LIN {X 86.419,Y -41.764,Z -98.944,A -90.000,B 90.000,C 0.000} C_DIS
LIN {X 86.321,Y -41.760,Z -99.036,A -90.000,B 90.000,C 0.000} C_DIS
LIN {X 86.213,Y -41.757,Z -99.132,A -90.000,B 90.000,C 0.000} C_DIS
LIN {X 85.903,Y -41.758,Z -99.390,A -90.000,B 90.000,C 0.000} C_DIS
LIN {X 85.446,Y -41.767,Z -99.745,A -90.000,B 90.000,C 0.000} C_DIS
LIN {X 85.305,Y -41.778,Z -99.859,A -90.000,B 90.000,C 0.000} C_DIS
LIN {X 85.131,Y -41.796,Z -99.993,A -90.000,B 90.000,C 0.000} C_DIS
LIN {X 84.957,Y -41.819,Z -100.115,A -90.000,B 90.000,C 0.000} C_DIS
LIN {X 84.802,Y -41.842,Z -100.215,A -90.000,B 90.000,C 0.000} C_DIS
LIN {X 84.683,Y -41.862,Z -100.286,A -90.000,B 90.000,C 0.000} C_DIS
LIN {X 84.481,Y -41.884,Z -100.395,A -90.000,B 90.000,C 0.000} C_DIS
LIN {X 84.221,Y -41.928,Z -100.537,A -90.000,B 90.000,C 0.000} C_DIS
LIN {X 84.067,Y -41.950,Z -100.619,A -90.000,B 90.000,C 0.000} C_DIS
LIN {X 83.579,Y -42.021,Z -100.876,A -90.000,B 90.000,C 0.000} C_DIS
LIN {X 83.391,Y -42.049,Z -100.970,A -90.000,B 90.000,C 0.000} C_DIS
LIN {X 83.264,Y -42.075,Z -101.035,A -90.000,B 90.000,C 0.000} C_DIS
LIN {X 82.879,Y -42.146,Z -101.260,A -90.000,B 90.000,C 0.000} C_DIS
LIN {X 82.672,Y -42.176,Z -101.400,A -90.000,B 90.000,C 0.000} C_DIS
LIN {X 82.594,Y -42.188,Z -101.451,A -90.000,B 90.000,C 0.000} C_DIS
LIN {X 82.374,Y -42.226,Z -101.578,A -90.000,B 90.000,C 0.000} C_DIS
LIN {X 82.222,Y -42.254,Z -101.660,A -90.000,B 90.000,C 0.000} C_DIS
LIN {X 82.012,Y -42.297,Z -101.771,A -90.000,B 90.000,C 0.000} C_DIS
LIN {X 81.894,Y -42.322,Z -101.825,A -90.000,B 90.000,C 0.000} C_DIS
LIN {X 81.742,Y -42.355,Z -101.888,A -90.000,B 90.000,C 0.000} C_DIS
LIN {X 81.659,Y -42.371,Z -101.920,A -90.000,B 90.000,C 0.000} C_DIS
LIN {X 81.529,Y -42.394,Z -101.964,A -90.000,B 90.000,C 0.000} C_DIS
LIN {X 81.072,Y -42.475,Z -102.099,A -90.000,B 90.000,C 0.000} C_DIS
LIN {X 81.028,Y -42.482,Z -102.115,A -90.000,B 90.000,C 0.000} C_DIS
LIN {X 80.881,Y -42.501,Z -102.170,A -90.000,B 90.000,C 0.000} C_DIS
LIN {X 80.690,Y -42.524,Z -102.247,A -90.000,B 90.000,C 0.000} C_DIS
LIN {X 80.320,Y -42.591,Z -102.396,A -90.000,B 90.000,C 0.000} C_DIS
LIN {X 79.816,Y -42.684,Z -102.594,A -90.000,B 90.000,C 0.000} C_DIS
LIN {X 79.637,Y -42.717,Z -102.663,A -90.000,B 90.000,C 0.000} C_DIS
LIN {X 79.531,Y -42.736,Z -102.698,A -90.000,B 90.000,C 0.000} C_DIS
LIN {X 79.408,Y -42.759,Z -102.750,A -90.000,B 90.000,C 0.000} C_DIS
LIN {X 79.279,Y -42.782,Z -102.801,A -90.000,B 90.000,C 0.000} C_DIS
LIN {X 79.059,Y -42.822,Z -102.874,A -90.000,B 90.000,C 0.000} C_DIS
LIN {X 78.928,Y -42.846,Z -102.910,A -90.000,B 90.000,C 0.000} C_DIS
LIN {X 78.902,Y -42.851,Z -102.916,A -90.000,B 90.000,C 0.000} C_DIS
LIN {X 78.691,Y -42.870,Z -102.962,A -90.000,B 90.000,C 0.000} C_DIS
LIN {X 78.445,Y -42.891,Z -103.005,A -90.000,B 90.000,C 0.000} C_DIS
LIN {X 78.333,Y -42.900,Z -103.021,A -90.000,B 90.000,C 0.000} C_DIS
LIN {X 78.121,Y -42.912,Z -103.046,A -90.000,B 90.000,C 0.000} C_DIS
LIN {X 77.986,Y -42.919,Z -103.054,A -90.000,B 90.000,C 0.000} C_DIS
LIN {X 77.768,Y -42.931,Z -103.059,A -90.000,B 90.000,C 0.000} C_DIS
LIN {X 77.616,Y -42.940,Z -103.055,A -90.000,B 90.000,C 0.000} C_DIS
LIN {X 77.437,Y -42.949,Z -103.044,A -90.000,B 90.000,C 0.000} C_DIS
LIN {X 77.279,Y -42.957,Z -103.028,A -90.000,B 90.000,C 0.000} C_DIS
LIN {X 77.030,Y -42.970,Z -102.997,A -90.000,B 90.000,C 0.000} C_DIS
LIN {X 76.845,Y -42.979,Z -102.965,A -90.000,B 90.000,C 0.000} C_DIS
LIN {X 76.645,Y -42.989,Z -102.921,A -90.000,B 90.000,C 0.000} C_DIS
LIN {X 76.463,Y -43.002,Z -102.870,A -90.000,B 90.000,C 0.000} C_DIS
LIN {X 76.351,Y -43.011,Z -102.835,A -90.000,B 90.000,C 0.000} C_DIS
LIN {X 76.162,Y -43.012,Z -102.772,A -90.000,B 90.000,C 0.000} C_DIS
LIN {X 76.056,Y -43.009,Z -102.736,A -90.000,B 90.000,C 0.000} C_DIS
LIN {X 75.843,Y -42.992,Z -102.665,A -90.000,B 90.000,C 0.000} C_DIS
LIN {X 74.970,Y -42.921,Z -102.398,A -90.000,B 90.000,C 0.000} C_DIS
LIN {X 74.859,Y -42.912,Z -102.360,A -90.000,B 90.000,C 0.000} C_DIS
LIN {X 74.584,Y -42.889,Z -102.259,A -90.000,B 90.000,C 0.000} C_DIS
LIN {X 74.543,Y -42.886,Z -102.242,A -90.000,B 90.000,C 0.000} C_DIS
LIN {X 74.381,Y -42.876,Z -102.172,A -90.000,B 90.000,C 0.000} C_DIS
LIN {X 74.239,Y -42.869,Z -102.108,A -90.000,B 90.000,C 0.000} C_DIS
LIN {X 74.136,Y -42.863,Z -102.058,A -90.000,B 90.000,C 0.000} C_DIS
LIN {X 74.017,Y -42.853,Z -101.993,A -90.000,B 90.000,C 0.000} C_DIS
LIN {X 73.964,Y -42.845,Z -101.963,A -90.000,B 90.000,C 0.000} C_DIS
LIN {X 73.864,Y -42.826,Z -101.902,A -90.000,B 90.000,C 0.000} C_DIS
LIN {X 73.750,Y -42.803,Z -101.827,A -90.000,B 90.000,C 0.000} C_DIS
LIN {X 73.573,Y -42.769,Z -101.698,A -90.000,B 90.000,C 0.000} C_DIS
LIN {X 73.484,Y -42.751,Z -101.627,A -90.000,B 90.000,C 0.000} C_DIS
LIN {X 73.297,Y -42.714,Z -101.471,A -90.000,B 90.000,C 0.000} C_DIS
LIN {X 73.161,Y -42.687,Z -101.346,A -90.000,B 90.000,C 0.000} C_DIS
LIN {X 72.996,Y -42.667,Z -101.190,A -90.000,B 90.000,C 0.000} C_DIS
LIN {X 72.866,Y -42.653,Z -101.050,A -90.000,B 90.000,C 0.000} C_DIS
LIN {X 72.774,Y -42.643,Z -100.942,A -90.000,B 90.000,C 0.000} C_DIS
LIN {X 72.642,Y -42.630,Z -100.772,A -90.000,B 90.000,C 0.000} C_DIS
LIN {X 72.484,Y -42.614,Z -100.550,A -90.000,B 90.000,C 0.000} C_DIS
LIN {X 72.383,Y -42.593,Z -100.404,A -90.000,B 90.000,C 0.000} C_DIS
LIN {X 72.177,Y -42.562,Z -100.105,A -90.000,B 90.000,C 0.000} C_DIS
LIN {X 71.790,Y -42.499,Z -99.545,A -90.000,B 90.000,C 0.000} C_DIS
LIN {X 71.523,Y -42.475,Z -99.165,A -90.000,B 90.000,C 0.000} C_DIS
LIN {X 71.422,Y -42.463,Z -99.016,A -90.000,B 90.000,C 0.000} C_DIS
LIN {X 71.303,Y -42.445,Z -98.829,A -90.000,B 90.000,C 0.000} C_DIS
LIN {X 71.201,Y -42.433,Z -98.643,A -90.000,B 90.000,C 0.000} C_DIS
LIN {X 71.153,Y -42.427,Z -98.549,A -90.000,B 90.000,C 0.000} C_DIS
LIN {X 71.078,Y -42.425,Z -98.401,A -90.000,B 90.000,C 0.000} C_DIS
LIN {X 70.998,Y -42.425,Z -98.226,A -90.000,B 90.000,C 0.000} C_DIS
LIN {X 70.815,Y -42.432,Z -97.770,A -90.000,B 90.000,C 0.000} C_DIS
LIN {X 70.779,Y -42.432,Z -97.674,A -90.000,B 90.000,C 0.000} C_DIS
LIN {X 70.656,Y -42.433,Z -97.314,A -90.000,B 90.000,C 0.000} C_DIS
LIN {X 70.437,Y -42.452,Z -96.657,A -90.000,B 90.000,C 0.000} C_DIS
LIN {X 70.362,Y -42.461,Z -96.404,A -90.000,B 90.000,C 0.000} C_DIS
LIN {X 70.336,Y -42.466,Z -96.298,A -90.000,B 90.000,C 0.000} C_DIS
LIN {X 70.140,Y -42.513,Z -95.413,A -90.000,B 90.000,C 0.000} C_DIS
LIN {X 70.084,Y -42.529,Z -95.124,A -90.000,B 90.000,C 0.000} C_DIS
LIN {X 70.025,Y -42.541,Z -94.775,A -90.000,B 90.000,C 0.000} C_DIS
LIN {X 69.988,Y -42.553,Z -94.483,A -90.000,B 90.000,C 0.000} C_DIS
LIN {X 69.976,Y -42.558,Z -94.352,A -90.000,B 90.000,C 0.000} C_DIS
LIN {X 69.968,Y -42.565,Z -94.224,A -90.000,B 90.000,C 0.000} C_DIS
LIN {X 69.923,Y -42.630,Z -92.991,A -90.000,B 90.000,C 0.000} C_DIS
LIN {X 69.922,Y -42.635,Z -92.892,A -90.000,B 90.000,C 0.000} C_DIS
LIN {X 69.941,Y -42.665,Z -92.441,A -90.000,B 90.000,C 0.000} C_DIS
LIN {X 69.960,Y -42.678,Z -92.274,A -90.000,B 90.000,C 0.000} C_DIS
LIN {X 69.993,Y -42.698,Z -92.009,A -90.000,B 90.000,C 0.000} C_DIS
LIN {X 70.053,Y -42.716,Z -91.546,A -90.000,B 90.000,C 0.000} C_DIS
LIN {X 70.089,Y -42.724,Z -91.330,A -90.000,B 90.000,C 0.000} C_DIS
LIN {X 70.112,Y -42.729,Z -91.213,A -90.000,B 90.000,C 0.000} C_DIS
LIN {X 70.168,Y -42.740,Z -90.959,A -90.000,B 90.000,C 0.000} C_DIS
LIN {X 70.198,Y -42.746,Z -90.842,A -90.000,B 90.000,C 0.000} C_DIS
LIN {X 70.296,Y -42.764,Z -90.535,A -90.000,B 90.000,C 0.000} C_DIS
LIN {X 70.377,Y -42.779,Z -90.327,A -90.000,B 90.000,C 0.000} C_DIS
LIN {X 70.481,Y -42.797,Z -90.099,A -90.000,B 90.000,C 0.000} C_DIS
LIN {X 70.517,Y -42.803,Z -90.028,A -90.000,B 90.000,C 0.000} C_DIS
LIN {X 70.645,Y -42.810,Z -89.783,A -90.000,B 90.000,C 0.000} C_DIS
LIN {X 70.735,Y -42.814,Z -89.612,A -90.000,B 90.000,C 0.000} C_DIS
LIN {X 70.797,Y -42.814,Z -89.437,A -90.000,B 90.000,C 0.000} C_DIS
LIN {X 70.851,Y -42.816,Z -89.307,A -90.000,B 90.000,C 0.000} C_DIS
LIN {X 70.936,Y -42.819,Z -89.122,A -90.000,B 90.000,C 0.000} C_DIS
LIN {X 71.088,Y -42.826,Z -88.833,A -90.000,B 90.000,C 0.000} C_DIS
LIN {X 71.230,Y -42.834,Z -88.606,A -90.000,B 90.000,C 0.000} C_DIS
LIN {X 71.313,Y -42.840,Z -88.492,A -90.000,B 90.000,C 0.000} C_DIS
LIN {X 71.412,Y -42.842,Z -88.355,A -90.000,B 90.000,C 0.000} C_DIS
LIN {X 71.536,Y -42.839,Z -88.186,A -90.000,B 90.000,C 0.000} C_DIS
LIN {X 71.639,Y -42.833,Z -88.057,A -90.000,B 90.000,C 0.000} C_DIS
LIN {X 71.757,Y -42.823,Z -87.932,A -90.000,B 90.000,C 0.000} C_DIS
LIN {X 71.833,Y -42.817,Z -87.856,A -90.000,B 90.000,C 0.000} C_DIS
LIN {X 71.936,Y -42.813,Z -87.753,A -90.000,B 90.000,C 0.000} C_DIS
LIN {X 72.037,Y -42.810,Z -87.659,A -90.000,B 90.000,C 0.000} C_DIS
LIN {X 72.176,Y -42.806,Z -87.538,A -90.000,B 90.000,C 0.000} C_DIS
LIN {X 72.275,Y -42.804,Z -87.459,A -90.000,B 90.000,C 0.000} C_DIS
LIN {X 72.481,Y -42.801,Z -87.309,A -90.000,B 90.000,C 0.000} C_DIS
LIN {X 72.543,Y -42.798,Z -87.246,A -90.000,B 90.000,C 0.000} C_DIS
LIN {X 72.657,Y -42.789,Z -87.140,A -90.000,B 90.000,C 0.000} C_DIS
LIN {X 72.771,Y -42.774,Z -87.041,A -90.000,B 90.000,C 0.000} C_DIS
LIN {X 72.930,Y -42.742,Z -86.909,A -90.000,B 90.000,C 0.000} C_DIS
LIN {X 73.086,Y -42.723,Z -86.795,A -90.000,B 90.000,C 0.000} C_DIS
LIN {X 73.242,Y -42.706,Z -86.693,A -90.000,B 90.000,C 0.000} C_DIS
LIN {X 73.408,Y -42.689,Z -86.595,A -90.000,B 90.000,C 0.000} C_DIS
LIN {X 73.664,Y -42.663,Z -86.455,A -90.000,B 90.000,C 0.000} C_DIS
LIN {X 73.879,Y -42.638,Z -86.352,A -90.000,B 90.000,C 0.000} C_DIS
LIN {X 73.927,Y -42.632,Z -86.332,A -90.000,B 90.000,C 0.000} C_DIS
LIN {X 74.005,Y -42.618,Z -86.282,A -90.000,B 90.000,C 0.000} C_DIS
LIN {X 74.160,Y -42.587,Z -86.190,A -90.000,B 90.000,C 0.000} C_DIS
LIN {X 74.313,Y -42.558,Z -86.108,A -90.000,B 90.000,C 0.000} C_DIS
LIN {X 74.493,Y -42.526,Z -86.017,A -90.000,B 90.000,C 0.000} C_DIS
LIN {X 74.658,Y -42.509,Z -85.938,A -90.000,B 90.000,C 0.000} C_DIS
LIN {X 74.676,Y -42.507,Z -85.929,A -90.000,B 90.000,C 0.000} C_DIS
LIN {X 74.798,Y -42.473,Z -85.813,A -90.000,B 90.000,C 0.000} C_DIS
LIN {X 74.935,Y -42.429,Z -85.703,A -90.000,B 90.000,C 0.000} C_DIS
LIN {X 75.148,Y -42.363,Z -85.542,A -90.000,B 90.000,C 0.000} C_DIS
LIN {X 75.177,Y -42.354,Z -85.522,A -90.000,B 90.000,C 0.000} C_DIS
LIN {X 75.264,Y -42.338,Z -85.461,A -90.000,B 90.000,C 0.000} C_DIS
LIN {X 75.410,Y -42.300,Z -85.316,A -90.000,B 90.000,C 0.000} C_DIS
LIN {X 75.571,Y -42.258,Z -85.161,A -90.000,B 90.000,C 0.000} C_DIS
LIN {X 75.690,Y -42.229,Z -85.055,A -90.000,B 90.000,C 0.000} C_DIS
LIN {X 75.797,Y -42.203,Z -84.968,A -90.000,B 90.000,C 0.000} C_DIS
LIN {X 76.148,Y -42.117,Z -84.702,A -90.000,B 90.000,C 0.000} C_DIS
LIN {X 76.215,Y -42.096,Z -84.654,A -90.000,B 90.000,C 0.000} C_DIS
LIN {X 76.516,Y -42.039,Z -84.425,A -90.000,B 90.000,C 0.000} C_DIS
LIN {X 76.658,Y -42.014,Z -84.321,A -90.000,B 90.000,C 0.000} C_DIS
LIN {X 76.854,Y -41.992,Z -84.183,A -90.000,B 90.000,C 0.000} C_DIS
LIN {X 77.017,Y -41.966,Z -84.064,A -90.000,B 90.000,C 0.000} C_DIS
LIN {X 77.252,Y -41.934,Z -83.904,A -90.000,B 90.000,C 0.000} C_DIS
LIN {X 77.345,Y -41.922,Z -83.844,A -90.000,B 90.000,C 0.000} C_DIS
LIN {X 77.479,Y -41.906,Z -83.764,A -90.000,B 90.000,C 0.000} C_DIS
LIN {X 77.605,Y -41.891,Z -83.695,A -90.000,B 90.000,C 0.000} C_DIS
LIN {X 77.706,Y -41.883,Z -83.644,A -90.000,B 90.000,C 0.000} C_DIS
LIN {X 77.905,Y -41.872,Z -83.549,A -90.000,B 90.000,C 0.000} C_DIS
LIN {X 77.931,Y -41.871,Z -83.537,A -90.000,B 90.000,C 0.000} C_DIS
LIN {X 77.948,Y -41.869,Z -83.525,A -90.000,B 90.000,C 0.000} C_DIS
LIN {X 78.237,Y -41.828,Z -83.332,A -90.000,B 90.000,C 0.000} C_DIS
LIN {X 78.363,Y -41.822,Z -83.241,A -90.000,B 90.000,C 0.000} C_DIS
LIN {X 78.440,Y -41.812,Z -83.189,A -90.000,B 90.000,C 0.000} C_DIS
LIN {X 78.548,Y -41.801,Z -83.120,A -90.000,B 90.000,C 0.000} C_DIS
LIN {X 78.707,Y -41.785,Z -83.026,A -90.000,B 90.000,C 0.000} C_DIS
LIN {X 78.831,Y -41.773,Z -82.958,A -90.000,B 90.000,C 0.000} C_DIS
LIN {X 79.141,Y -41.753,Z -82.808,A -90.000,B 90.000,C 0.000} C_DIS
LIN {X 79.305,Y -41.746,Z -82.735,A -90.000,B 90.000,C 0.000} C_DIS
LIN {X 79.442,Y -41.741,Z -82.679,A -90.000,B 90.000,C 0.000} C_DIS
LIN {X 79.615,Y -41.737,Z -82.616,A -90.000,B 90.000,C 0.000} C_DIS
LIN {X 79.691,Y -41.741,Z -82.585,A -90.000,B 90.000,C 0.000} C_DIS
LIN {X 79.828,Y -41.750,Z -82.536,A -90.000,B 90.000,C 0.000} C_DIS
LIN {X 80.478,Y -41.803,Z -82.324,A -90.000,B 90.000,C 0.000} C_DIS
LIN {X 80.770,Y -41.866,Z -82.214,A -90.000,B 90.000,C 0.000} C_DIS
LIN {X 80.716,Y -41.780,Z -82.049,A -90.000,B 90.000,C 0.000} C_DIS
LIN {X 80.609,Y -41.586,Z -81.693,A -90.000,B 90.000,C 0.000} C_DIS
LIN {X 80.594,Y -41.556,Z -81.636,A -90.000,B 90.000,C 0.000} C_DIS
LIN {X 80.558,Y -41.492,Z -81.495,A -90.000,B 90.000,C 0.000} C_DIS
LIN {X 80.524,Y -41.422,Z -81.332,A -90.000,B 90.000,C 0.000} C_DIS
LIN {X 80.480,Y -41.308,Z -81.051,A -90.000,B 90.000,C 0.000} C_DIS
LIN {X 80.480,Y -60.000,Z -81.051,A -90.000,B 90.000,C 0.000} C_DIS
LIN {X 84.763,Y -60.000,Z -102.385,A -90.000,B 90.000,C 0.000} C_DIS
LIN {X 84.763,Y -41.308,Z -102.385,A -90.000,B 90.000,C 0.000} C_DIS
LIN {X 84.387,Y -41.438,Z -102.611,A -90.000,B 90.000,C 0.000} C_DIS
LIN {X 84.107,Y -41.530,Z -102.766,A -90.000,B 90.000,C 0.000} C_DIS
LIN {X 83.918,Y -41.589,Z -102.884,A -90.000,B 90.000,C 0.000} C_DIS
LIN {X 83.845,Y -41.612,Z -102.929,A -90.000,B 90.000,C 0.000} C_DIS
LIN {X 83.619,Y -41.685,Z -103.093,A -90.000,B 90.000,C 0.000} C_DIS
LIN {X 83.508,Y -41.722,Z -103.167,A -90.000,B 90.000,C 0.000} C_DIS
LIN {X 83.248,Y -41.806,Z -103.327,A -90.000,B 90.000,C 0.000} C_DIS
LIN {X 83.028,Y -41.878,Z -103.452,A -90.000,B 90.000,C 0.000} C_DIS
LIN {X 82.852,Y -41.935,Z -103.549,A -90.000,B 90.000,C 0.000} C_DIS
LIN {X 82.666,Y -41.994,Z -103.641,A -90.000,B 90.000,C 0.000} C_DIS
LIN {X 82.443,Y -42.066,Z -103.739,A -90.000,B 90.000,C 0.000} C_DIS
LIN {X 82.257,Y -42.125,Z -103.812,A -90.000,B 90.000,C 0.000} C_DIS
LIN {X 82.058,Y -42.189,Z -103.882,A -90.000,B 90.000,C 0.000} C_DIS
LIN {X 81.674,Y -42.311,Z -104.000,A -90.000,B 90.000,C 0.000} C_DIS
LIN {X 81.576,Y -42.341,Z -104.039,A -90.000,B 90.000,C 0.000} C_DIS
LIN {X 81.153,Y -42.469,Z -104.213,A -90.000,B 90.000,C 0.000} C_DIS
LIN {X 80.593,Y -42.578,Z -104.435,A -90.000,B 90.000,C 0.000} C_DIS
LIN {X 80.338,Y -42.617,Z -104.534,A -90.000,B 90.000,C 0.000} C_DIS
LIN {X 80.222,Y -42.634,Z -104.574,A -90.000,B 90.000,C 0.000} C_DIS
LIN {X 80.146,Y -42.646,Z -104.606,A -90.000,B 90.000,C 0.000} C_DIS
LIN {X 79.982,Y -42.670,Z -104.670,A -90.000,B 90.000,C 0.000} C_DIS
LIN {X 79.787,Y -42.699,Z -104.736,A -90.000,B 90.000,C 0.000} C_DIS
LIN {X 79.672,Y -42.716,Z -104.775,A -90.000,B 90.000,C 0.000} C_DIS
LIN {X 79.574,Y -42.731,Z -104.804,A -90.000,B 90.000,C 0.000} C_DIS
LIN {X 79.363,Y -42.762,Z -104.860,A -90.000,B 90.000,C 0.000} C_DIS
LIN {X 79.032,Y -42.810,Z -104.932,A -90.000,B 90.000,C 0.000} C_DIS
LIN {X 78.721,Y -42.854,Z -104.986,A -90.000,B 90.000,C 0.000} C_DIS
LIN {X 78.565,Y -42.876,Z -105.007,A -90.000,B 90.000,C 0.000} C_DIS
LIN {X 78.354,Y -42.905,Z -105.032,A -90.000,B 90.000,C 0.000} C_DIS
LIN {X 78.197,Y -42.926,Z -105.045,A -90.000,B 90.000,C 0.000} C_DIS
LIN {X 77.989,Y -42.944,Z -105.054,A -90.000,B 90.000,C 0.000} C_DIS
LIN {X 77.744,Y -42.965,Z -105.059,A -90.000,B 90.000,C 0.000} C_DIS
LIN {X 77.685,Y -42.970,Z -105.058,A -90.000,B 90.000,C 0.000} C_DIS
LIN {X 77.487,Y -42.973,Z -105.051,A -90.000,B 90.000,C 0.000} C_DIS
LIN {X 77.238,Y -42.975,Z -105.033,A -90.000,B 90.000,C 0.000} C_DIS
LIN {X 77.035,Y -42.976,Z -105.013,A -90.000,B 90.000,C 0.000} C_DIS
LIN {X 76.786,Y -42.978,Z -104.982,A -90.000,B 90.000,C 0.000} C_DIS
LIN {X 76.609,Y -42.979,Z -104.954,A -90.000,B 90.000,C 0.000} C_DIS
LIN {X 76.421,Y -42.981,Z -104.919,A -90.000,B 90.000,C 0.000} C_DIS
LIN {X 76.220,Y -42.983,Z -104.875,A -90.000,B 90.000,C 0.000} C_DIS
LIN {X 76.105,Y -42.984,Z -104.847,A -90.000,B 90.000,C 0.000} C_DIS
LIN {X 75.863,Y -42.986,Z -104.778,A -90.000,B 90.000,C 0.000} C_DIS
LIN {X 75.716,Y -42.988,Z -104.731,A -90.000,B 90.000,C 0.000} C_DIS
LIN {X 75.328,Y -42.991,Z -104.602,A -90.000,B 90.000,C 0.000} C_DIS
LIN {X 75.224,Y -42.988,Z -104.567,A -90.000,B 90.000,C 0.000} C_DIS
LIN {X 74.754,Y -42.946,Z -104.423,A -90.000,B 90.000,C 0.000} C_DIS
LIN {X 74.542,Y -42.914,Z -104.358,A -90.000,B 90.000,C 0.000} C_DIS
LIN {X 74.387,Y -42.894,Z -104.311,A -90.000,B 90.000,C 0.000} C_DIS
LIN {X 74.174,Y -42.868,Z -104.239,A -90.000,B 90.000,C 0.000} C_DIS
LIN {X 73.900,Y -42.833,Z -104.138,A -90.000,B 90.000,C 0.000} C_DIS
LIN {X 73.768,Y -42.817,Z -104.084,A -90.000,B 90.000,C 0.000} C_DIS
LIN {X 73.490,Y -42.782,Z -103.962,A -90.000,B 90.000,C 0.000} C_DIS
LIN {X 73.366,Y -42.767,Z -103.904,A -90.000,B 90.000,C 0.000} C_DIS
LIN {X 73.186,Y -42.744,Z -103.814,A -90.000,B 90.000,C 0.000} C_DIS
LIN {X 73.071,Y -42.729,Z -103.751,A -90.000,B 90.000,C 0.000} C_DIS
LIN {X 72.940,Y -42.703,Z -103.675,A -90.000,B 90.000,C 0.000} C_DIS
LIN {X 72.792,Y -42.672,Z -103.583,A -90.000,B 90.000,C 0.000} C_DIS
LIN {X 72.662,Y -42.644,Z -103.497,A -90.000,B 90.000,C 0.000} C_DIS
LIN {X 72.600,Y -42.626,Z -103.454,A -90.000,B 90.000,C 0.000} C_DIS
LIN {X 72.362,Y -42.565,Z -103.277,A -90.000,B 90.000,C 0.000} C_DIS
LIN {X 72.235,Y -42.532,Z -103.174,A -90.000,B 90.000,C 0.000} C_DIS
LIN {X 71.999,Y -42.469,Z -102.972,A -90.000,B 90.000,C 0.000} C_DIS
LIN {X 71.796,Y -42.414,Z -102.782,A -90.000,B 90.000,C 0.000} C_DIS
LIN {X 71.661,Y -42.377,Z -102.651,A -90.000,B 90.000,C 0.000} C_DIS
LIN {X 71.562,Y -42.359,Z -102.549,A -90.000,B 90.000,C 0.000} C_DIS
LIN {X 71.435,Y -42.335,Z -102.410,A -90.000,B 90.000,C 0.000} C_DIS
LIN {X 71.374,Y -42.316,Z -102.338,A -90.000,B 90.000,C 0.000} C_DIS
LIN {X 71.244,Y -42.272,Z -102.174,A -90.000,B 90.000,C 0.000} C_DIS
LIN {X 71.093,Y -42.222,Z -101.970,A -90.000,B 90.000,C 0.000} C_DIS
LIN {X 70.878,Y -42.145,Z -101.648,A -90.000,B 90.000,C 0.000} C_DIS
LIN {X 70.336,Y -42.018,Z -100.847,A -90.000,B 90.000,C 0.000} C_DIS
LIN {X 70.232,Y -41.998,Z -100.694,A -90.000,B 90.000,C 0.000} C_DIS
LIN {X 69.984,Y -41.942,Z -100.327,A -90.000,B 90.000,C 0.000} C_DIS
LIN {X 69.816,Y -41.905,Z -100.069,A -90.000,B 90.000,C 0.000} C_DIS
LIN {X 69.720,Y -41.884,Z -99.914,A -90.000,B 90.000,C 0.000} C_DIS
LIN {X 69.649,Y -41.877,Z -99.798,A -90.000,B 90.000,C 0.000} C_DIS
LIN {X 69.506,Y -41.864,Z -99.541,A -90.000,B 90.000,C 0.000} C_DIS
LIN {X 69.389,Y -41.857,Z -99.308,A -90.000,B 90.000,C 0.000} C_DIS
LIN {X 69.329,Y -41.854,Z -99.184,A -90.000,B 90.000,C 0.000} C_DIS
LIN {X 69.241,Y -41.855,Z -98.992,A -90.000,B 90.000,C 0.000} C_DIS
LIN {X 69.032,Y -41.868,Z -98.480,A -90.000,B 90.000,C 0.000} C_DIS
LIN {X 68.941,Y -41.878,Z -98.238,A -90.000,B 90.000,C 0.000} C_DIS
LIN {X 68.813,Y -41.894,Z -97.875,A -90.000,B 90.000,C 0.000} C_DIS
LIN {X 68.580,Y -41.929,Z -97.184,A -90.000,B 90.000,C 0.000} C_DIS
LIN {X 68.504,Y -41.945,Z -96.932,A -90.000,B 90.000,C 0.000} C_DIS
LIN {X 68.464,Y -41.956,Z -96.784,A -90.000,B 90.000,C 0.000} C_DIS
LIN {X 68.439,Y -41.964,Z -96.684,A -90.000,B 90.000,C 0.000} C_DIS
LIN {X 68.241,Y -42.036,Z -95.823,A -90.000,B 90.000,C 0.000} C_DIS
LIN {X 68.169,Y -42.067,Z -95.472,A -90.000,B 90.000,C 0.000} C_DIS
LIN {X 68.101,Y -42.090,Z -95.083,A -90.000,B 90.000,C 0.000} C_DIS
LIN {X 68.069,Y -42.106,Z -94.858,A -90.000,B 90.000,C 0.000} C_DIS
LIN {X 68.042,Y -42.120,Z -94.646,A -90.000,B 90.000,C 0.000} C_DIS
LIN {X 68.024,Y -42.133,Z -94.451,A -90.000,B 90.000,C 0.000} C_DIS
LIN {X 68.011,Y -42.149,Z -94.232,A -90.000,B 90.000,C 0.000} C_DIS
LIN {X 67.962,Y -42.239,Z -92.992,A -90.000,B 90.000,C 0.000} C_DIS
LIN {X 67.960,Y -42.247,Z -92.880,A -90.000,B 90.000,C 0.000} C_DIS
LIN {X 67.962,Y -42.257,Z -92.773,A -90.000,B 90.000,C 0.000} C_DIS
LIN {X 67.982,Y -42.281,Z -92.329,A -90.000,B 90.000,C 0.000} C_DIS
LIN {X 67.993,Y -42.289,Z -92.187,A -90.000,B 90.000,C 0.000} C_DIS
LIN {X 68.048,Y -42.321,Z -91.738,A -90.000,B 90.000,C 0.000} C_DIS
LIN {X 68.105,Y -42.353,Z -91.278,A -90.000,B 90.000,C 0.000} C_DIS
LIN {X 68.159,Y -42.380,Z -90.933,A -90.000,B 90.000,C 0.000} C_DIS
LIN {X 68.188,Y -42.393,Z -90.781,A -90.000,B 90.000,C 0.000} C_DIS
LIN {X 68.244,Y -42.416,Z -90.518,A -90.000,B 90.000,C 0.000} C_DIS
LIN {X 68.287,Y -42.429,Z -90.342,A -90.000,B 90.000,C 0.000} C_DIS
LIN {X 68.321,Y -42.439,Z -90.222,A -90.000,B 90.000,C 0.000} C_DIS
LIN {X 68.357,Y -42.447,Z -90.110,A -90.000,B 90.000,C 0.000} C_DIS
LIN {X 68.417,Y -42.457,Z -89.923,A -90.000,B 90.000,C 0.000} C_DIS
LIN {X 68.460,Y -42.464,Z -89.802,A -90.000,B 90.000,C 0.000} C_DIS
LIN {X 68.562,Y -42.480,Z -89.542,A -90.000,B 90.000,C 0.000} C_DIS
LIN {X 68.689,Y -42.502,Z -89.261,A -90.000,B 90.000,C 0.000} C_DIS
LIN {X 68.762,Y -42.514,Z -89.114,A -90.000,B 90.000,C 0.000} C_DIS
LIN {X 68.917,Y -42.540,Z -88.812,A -90.000,B 90.000,C 0.000} C_DIS
LIN {X 68.972,Y -42.549,Z -88.663,A -90.000,B 90.000,C 0.000} C_DIS
LIN {X 69.050,Y -42.562,Z -88.474,A -90.000,B 90.000,C 0.000} C_DIS
LIN {X 69.136,Y -42.576,Z -88.284,A -90.000,B 90.000,C 0.000} C_DIS
LIN {X 69.205,Y -42.588,Z -88.145,A -90.000,B 90.000,C 0.000} C_DIS
LIN {X 69.273,Y -42.593,Z -88.017,A -90.000,B 90.000,C 0.000} C_DIS
LIN {X 69.343,Y -42.595,Z -87.885,A -90.000,B 90.000,C 0.000} C_DIS
LIN {X 69.403,Y -42.597,Z -87.780,A -90.000,B 90.000,C 0.000} C_DIS
LIN {X 69.592,Y -42.605,Z -87.483,A -90.000,B 90.000,C 0.000} C_DIS
LIN {X 69.937,Y -42.622,Z -87.004,A -90.000,B 90.000,C 0.000} C_DIS
LIN {X 70.104,Y -42.631,Z -86.791,A -90.000,B 90.000,C 0.000} C_DIS
LIN {X 70.188,Y -42.635,Z -86.695,A -90.000,B 90.000,C 0.000} C_DIS
LIN {X 70.306,Y -42.639,Z -86.569,A -90.000,B 90.000,C 0.000} C_DIS
LIN {X 70.419,Y -42.638,Z -86.454,A -90.000,B 90.000,C 0.000} C_DIS
LIN {X 70.528,Y -42.634,Z -86.345,A -90.000,B 90.000,C 0.000} C_DIS
LIN {X 70.665,Y -42.623,Z -86.215,A -90.000,B 90.000,C 0.000} C_DIS
LIN {X 70.911,Y -42.598,Z -86.003,A -90.000,B 90.000,C 0.000} C_DIS
LIN {X 71.029,Y -42.592,Z -85.909,A -90.000,B 90.000,C 0.000} C_DIS
LIN {X 71.185,Y -42.584,Z -85.793,A -90.000,B 90.000,C 0.000} C_DIS
LIN {X 71.344,Y -42.572,Z -85.647,A -90.000,B 90.000,C 0.000} C_DIS
LIN {X 71.621,Y -42.553,Z -85.408,A -90.000,B 90.000,C 0.000} C_DIS
LIN {X 71.745,Y -42.539,Z -85.311,A -90.000,B 90.000,C 0.000} C_DIS
LIN {X 71.813,Y -42.527,Z -85.262,A -90.000,B 90.000,C 0.000} C_DIS
LIN {X 71.979,Y -42.495,Z -85.145,A -90.000,B 90.000,C 0.000} C_DIS
LIN {X 72.204,Y -42.452,Z -85.003,A -90.000,B 90.000,C 0.000} C_DIS
LIN {X 72.294,Y -42.433,Z -84.951,A -90.000,B 90.000,C 0.000} C_DIS
LIN {X 72.438,Y -42.410,Z -84.868,A -90.000,B 90.000,C 0.000} C_DIS
LIN {X 72.724,Y -42.369,Z -84.714,A -90.000,B 90.000,C 0.000} C_DIS
LIN {X 72.946,Y -42.339,Z -84.608,A -90.000,B 90.000,C 0.000} C_DIS
LIN {X 73.031,Y -42.325,Z -84.557,A -90.000,B 90.000,C 0.000} C_DIS
LIN {X 73.163,Y -42.295,Z -84.481,A -90.000,B 90.000,C 0.000} C_DIS
LIN {X 73.334,Y -42.246,Z -84.393,A -90.000,B 90.000,C 0.000} C_DIS
LIN {X 73.516,Y -42.200,Z -84.302,A -90.000,B 90.000,C 0.000} C_DIS
LIN {X 73.684,Y -42.145,Z -84.169,A -90.000,B 90.000,C 0.000} C_DIS
LIN {X 73.895,Y -42.078,Z -84.010,A -90.000,B 90.000,C 0.000} C_DIS
LIN {X 73.950,Y -42.061,Z -83.969,A -90.000,B 90.000,C 0.000} C_DIS
LIN {X 74.173,Y -41.977,Z -83.759,A -90.000,B 90.000,C 0.000} C_DIS
LIN {X 74.286,Y -41.935,Z -83.660,A -90.000,B 90.000,C 0.000} C_DIS
LIN {X 74.398,Y -41.886,Z -83.567,A -90.000,B 90.000,C 0.000} C_DIS
LIN {X 74.505,Y -41.841,Z -83.485,A -90.000,B 90.000,C 0.000} C_DIS
LIN {X 74.865,Y -41.696,Z -83.226,A -90.000,B 90.000,C 0.000} C_DIS
LIN {X 75.054,Y -41.636,Z -83.089,A -90.000,B 90.000,C 0.000} C_DIS
LIN {X 75.354,Y -41.517,Z -82.882,A -90.000,B 90.000,C 0.000} C_DIS
LIN {X 75.463,Y -41.475,Z -82.811,A -90.000,B 90.000,C 0.000} C_DIS
LIN {X 75.711,Y -41.376,Z -82.661,A -90.000,B 90.000,C 0.000} C_DIS
LIN {X 75.836,Y -41.337,Z -82.578,A -90.000,B 90.000,C 0.000} C_DIS
LIN {X 75.927,Y -41.308,Z -82.521,A -90.000,B 90.000,C 0.000} C_DIS
LIN {X 75.927,Y -60.000,Z -82.521,A -90.000,B 90.000,C 0.000} C_DIS
LIN {X 66.778,Y -60.000,Z -97.793,A -90.000,B 90.000,C 0.000} C_DIS
LIN {X 66.778,Y -41.308,Z -97.793,A -90.000,B 90.000,C 0.000} C_DIS
LIN {X 66.747,Y -41.315,Z -97.698,A -90.000,B 90.000,C 0.000} C_DIS
LIN {X 66.652,Y -41.338,Z -97.382,A -90.000,B 90.000,C 0.000} C_DIS
LIN {X 66.579,Y -41.362,Z -97.107,A -90.000,B 90.000,C 0.000} C_DIS
LIN {X 66.492,Y -41.396,Z -96.733,A -90.000,B 90.000,C 0.000} C_DIS
LIN {X 66.410,Y -41.427,Z -96.379,A -90.000,B 90.000,C 0.000} C_DIS
LIN {X 66.361,Y -41.441,Z -96.157,A -90.000,B 90.000,C 0.000} C_DIS
LIN {X 66.283,Y -41.470,Z -95.767,A -90.000,B 90.000,C 0.000} C_DIS
LIN {X 66.202,Y -41.506,Z -95.310,A -90.000,B 90.000,C 0.000} C_DIS
LIN {X 66.151,Y -41.537,Z -94.955,A -90.000,B 90.000,C 0.000} C_DIS
LIN {X 66.129,Y -41.553,Z -94.787,A -90.000,B 90.000,C 0.000} C_DIS
LIN {X 66.106,Y -41.577,Z -94.554,A -90.000,B 90.000,C 0.000} C_DIS
LIN {X 66.088,Y -41.605,Z -94.306,A -90.000,B 90.000,C 0.000} C_DIS
LIN {X 66.061,Y -41.664,Z -93.798,A -90.000,B 90.000,C 0.000} C_DIS
LIN {X 66.048,Y -41.688,Z -93.481,A -90.000,B 90.000,C 0.000} C_DIS
LIN {X 66.044,Y -41.695,Z -93.365,A -90.000,B 90.000,C 0.000} C_DIS
LIN {X 66.033,Y -41.708,Z -93.031,A -90.000,B 90.000,C 0.000} C_DIS
LIN {X 66.032,Y -41.720,Z -92.802,A -90.000,B 90.000,C 0.000} C_DIS
LIN {X 66.036,Y -41.728,Z -92.655,A -90.000,B 90.000,C 0.000} C_DIS
LIN {X 66.060,Y -41.762,Z -92.141,A -90.000,B 90.000,C 0.000} C_DIS
LIN {X 66.083,Y -41.783,Z -91.877,A -90.000,B 90.000,C 0.000} C_DIS
LIN {X 66.187,Y -41.859,Z -91.002,A -90.000,B 90.000,C 0.000} C_DIS
LIN {X 66.260,Y -41.898,Z -90.530,A -90.000,B 90.000,C 0.000} C_DIS
LIN {X 66.302,Y -41.917,Z -90.317,A -90.000,B 90.000,C 0.000} C_DIS
LIN {X 66.365,Y -41.941,Z -90.025,A -90.000,B 90.000,C 0.000} C_DIS
LIN {X 66.426,Y -41.963,Z -89.779,A -90.000,B 90.000,C 0.000} C_DIS
LIN {X 66.476,Y -41.981,Z -89.601,A -90.000,B 90.000,C 0.000} C_DIS
LIN {X 66.585,Y -42.019,Z -89.251,A -90.000,B 90.000,C 0.000} C_DIS
LIN {X 66.650,Y -42.040,Z -89.065,A -90.000,B 90.000,C 0.000} C_DIS
LIN {X 66.748,Y -42.073,Z -88.805,A -90.000,B 90.000,C 0.000} C_DIS
LIN {X 66.788,Y -42.086,Z -88.707,A -90.000,B 90.000,C 0.000} C_DIS
LIN {X 66.849,Y -42.107,Z -88.567,A -90.000,B 90.000,C 0.000} C_DIS
LIN {X 66.947,Y -42.137,Z -88.349,A -90.000,B 90.000,C 0.000} C_DIS
LIN {X 67.024,Y -42.153,Z -88.192,A -90.000,B 90.000,C 0.000} C_DIS
LIN {X 67.124,Y -42.172,Z -87.996,A -90.000,B 90.000,C 0.000} C_DIS
LIN {X 67.165,Y -42.180,Z -87.890,A -90.000,B 90.000,C 0.000} C_DIS
LIN {X 67.269,Y -42.197,Z -87.640,A -90.000,B 90.000,C 0.000} C_DIS
LIN {X 67.387,Y -42.216,Z -87.384,A -90.000,B 90.000,C 0.000} C_DIS
LIN {X 67.536,Y -42.243,Z -87.089,A -90.000,B 90.000,C 0.000} C_DIS
LIN {X 67.640,Y -42.261,Z -86.890,A -90.000,B 90.000,C 0.000} C_DIS
LIN {X 67.751,Y -42.282,Z -86.698,A -90.000,B 90.000,C 0.000} C_DIS
LIN {X 67.865,Y -42.308,Z -86.512,A -90.000,B 90.000,C 0.000} C_DIS
LIN {X 67.967,Y -42.318,Z -86.352,A -90.000,B 90.000,C 0.000} C_DIS
LIN {X 68.160,Y -42.338,Z -86.081,A -90.000,B 90.000,C 0.000} C_DIS
LIN {X 68.382,Y -42.349,Z -85.776,A -90.000,B 90.000,C 0.000} C_DIS
LIN {X 68.549,Y -42.358,Z -85.563,A -90.000,B 90.000,C 0.000} C_DIS
LIN {X 68.617,Y -42.362,Z -85.480,A -90.000,B 90.000,C 0.000} C_DIS
LIN {X 68.743,Y -42.371,Z -85.337,A -90.000,B 90.000,C 0.000} C_DIS
LIN {X 68.857,Y -42.379,Z -85.215,A -90.000,B 90.000,C 0.000} C_DIS
LIN {X 69.157,Y -42.408,Z -84.906,A -90.000,B 90.000,C 0.000} C_DIS
LIN {X 69.294,Y -42.415,Z -84.774,A -90.000,B 90.000,C 0.000} C_DIS
LIN {X 69.401,Y -42.417,Z -84.678,A -90.000,B 90.000,C 0.000} C_DIS
LIN {X 69.541,Y -42.412,Z -84.556,A -90.000,B 90.000,C 0.000} C_DIS
LIN {X 69.679,Y -42.402,Z -84.440,A -90.000,B 90.000,C 0.000} C_DIS
LIN {X 69.840,Y -42.384,Z -84.315,A -90.000,B 90.000,C 0.000} C_DIS
LIN {X 69.907,Y -42.376,Z -84.265,A -90.000,B 90.000,C 0.000} C_DIS
LIN {X 70.039,Y -42.359,Z -84.146,A -90.000,B 90.000,C 0.000} C_DIS
LIN {X 70.374,Y -42.326,Z -83.862,A -90.000,B 90.000,C 0.000} C_DIS
LIN {X 70.556,Y -42.310,Z -83.719,A -90.000,B 90.000,C 0.000} C_DIS
LIN {X 70.703,Y -42.299,Z -83.612,A -90.000,B 90.000,C 0.000} C_DIS
LIN {X 70.837,Y -42.283,Z -83.517,A -90.000,B 90.000,C 0.000} C_DIS
LIN {X 71.163,Y -42.227,Z -83.310,A -90.000,B 90.000,C 0.000} C_DIS
LIN {X 71.302,Y -42.201,Z -83.230,A -90.000,B 90.000,C 0.000} C_DIS
LIN {X 71.547,Y -42.134,Z -83.097,A -90.000,B 90.000,C 0.000} C_DIS
LIN {X 71.756,Y -42.091,Z -82.986,A -90.000,B 90.000,C 0.000} C_DIS
LIN {X 71.836,Y -42.075,Z -82.947,A -90.000,B 90.000,C 0.000} C_DIS
LIN {X 71.976,Y -42.049,Z -82.881,A -90.000,B 90.000,C 0.000} C_DIS
LIN {X 72.182,Y -42.005,Z -82.762,A -90.000,B 90.000,C 0.000} C_DIS
LIN {X 72.344,Y -41.967,Z -82.677,A -90.000,B 90.000,C 0.000} C_DIS
LIN {X 72.399,Y -41.951,Z -82.649,A -90.000,B 90.000,C 0.000} C_DIS
LIN {X 72.635,Y -41.869,Z -82.470,A -90.000,B 90.000,C 0.000} C_DIS
LIN {X 72.752,Y -41.819,Z -82.360,A -90.000,B 90.000,C 0.000} C_DIS
LIN {X 72.818,Y -41.783,Z -82.301,A -90.000,B 90.000,C 0.000} C_DIS
LIN {X 72.909,Y -41.736,Z -82.223,A -90.000,B 90.000,C 0.000} C_DIS
LIN {X 73.124,Y -41.642,Z -82.045,A -90.000,B 90.000,C 0.000} C_DIS
LIN {X 73.279,Y -41.577,Z -81.927,A -90.000,B 90.000,C 0.000} C_DIS
LIN {X 73.499,Y -41.489,Z -81.769,A -90.000,B 90.000,C 0.000} C_DIS
LIN {X 73.886,Y -41.308,Z -81.499,A -90.000,B 90.000,C 0.000} C_DIS
LIN {X 73.886,Y -60.000,Z -81.499,A -90.000,B 90.000,C 0.000} C_DIS
LIN {X 64.566,Y -60.000,Z -89.413,A -90.000,B 90.000,C 0.000} C_DIS
LIN {X 64.566,Y -41.308,Z -89.413,A -90.000,B 90.000,C 0.000} C_DIS
LIN {X 64.618,Y -41.330,Z -89.204,A -90.000,B 90.000,C 0.000} C_DIS
LIN {X 64.682,Y -41.357,Z -88.975,A -90.000,B 90.000,C 0.000} C_DIS
LIN {X 64.808,Y -41.410,Z -88.565,A -90.000,B 90.000,C 0.000} C_DIS
LIN {X 64.892,Y -41.438,Z -88.324,A -90.000,B 90.000,C 0.000} C_DIS
LIN {X 65.031,Y -41.479,Z -87.966,A -90.000,B 90.000,C 0.000} C_DIS
LIN {X 65.132,Y -41.516,Z -87.728,A -90.000,B 90.000,C 0.000} C_DIS
LIN {X 65.252,Y -41.559,Z -87.458,A -90.000,B 90.000,C 0.000} C_DIS
LIN {X 65.389,Y -41.609,Z -87.169,A -90.000,B 90.000,C 0.000} C_DIS
LIN {X 65.527,Y -41.660,Z -86.817,A -90.000,B 90.000,C 0.000} C_DIS
LIN {X 65.631,Y -41.696,Z -86.580,A -90.000,B 90.000,C 0.000} C_DIS
LIN {X 65.683,Y -41.712,Z -86.466,A -90.000,B 90.000,C 0.000} C_DIS
LIN {X 65.882,Y -41.758,Z -86.071,A -90.000,B 90.000,C 0.000} C_DIS
LIN {X 65.941,Y -41.773,Z -85.956,A -90.000,B 90.000,C 0.000} C_DIS
LIN {X 66.092,Y -41.809,Z -85.687,A -90.000,B 90.000,C 0.000} C_DIS
LIN {X 66.349,Y -41.873,Z -85.264,A -90.000,B 90.000,C 0.000} C_DIS
LIN {X 66.470,Y -41.904,Z -85.085,A -90.000,B 90.000,C 0.000} C_DIS
LIN {X 66.693,Y -41.960,Z -84.761,A -90.000,B 90.000,C 0.000} C_DIS
LIN {X 66.800,Y -41.990,Z -84.607,A -90.000,B 90.000,C 0.000} C_DIS
LIN {X 66.879,Y -42.010,Z -84.500,A -90.000,B 90.000,C 0.000} C_DIS
LIN {X 66.990,Y -42.023,Z -84.356,A -90.000,B 90.000,C 0.000} C_DIS
LIN {X 67.146,Y -42.037,Z -84.165,A -90.000,B 90.000,C 0.000} C_DIS
LIN {X 67.307,Y -42.052,Z -83.982,A -90.000,B 90.000,C 0.000} C_DIS
LIN {X 67.455,Y -42.066,Z -83.823,A -90.000,B 90.000,C 0.000} C_DIS
LIN {X 67.791,Y -42.099,Z -83.478,A -90.000,B 90.000,C 0.000} C_DIS
LIN {X 67.974,Y -42.118,Z -83.302,A -90.000,B 90.000,C 0.000} C_DIS
LIN {X 68.009,Y -42.121,Z -83.269,A -90.000,B 90.000,C 0.000} C_DIS
LIN {X 68.279,Y -42.155,Z -83.025,A -90.000,B 90.000,C 0.000} C_DIS
LIN {X 68.391,Y -42.163,Z -82.928,A -90.000,B 90.000,C 0.000} C_DIS
LIN {X 68.525,Y -42.166,Z -82.820,A -90.000,B 90.000,C 0.000} C_DIS
LIN {X 68.640,Y -42.163,Z -82.729,A -90.000,B 90.000,C 0.000} C_DIS
LIN {X 68.739,Y -42.156,Z -82.640,A -90.000,B 90.000,C 0.000} C_DIS
LIN {X 68.808,Y -42.151,Z -82.581,A -90.000,B 90.000,C 0.000} C_DIS
LIN {X 68.944,Y -42.134,Z -82.466,A -90.000,B 90.000,C 0.000} C_DIS
LIN {X 69.136,Y -42.100,Z -82.307,A -90.000,B 90.000,C 0.000} C_DIS
LIN {X 69.258,Y -42.080,Z -82.213,A -90.000,B 90.000,C 0.000} C_DIS
LIN {X 69.376,Y -42.067,Z -82.122,A -90.000,B 90.000,C 0.000} C_DIS
LIN {X 69.635,Y -42.039,Z -81.938,A -90.000,B 90.000,C 0.000} C_DIS
LIN {X 69.744,Y -42.027,Z -81.862,A -90.000,B 90.000,C 0.000} C_DIS
LIN {X 70.005,Y -42.000,Z -81.693,A -90.000,B 90.000,C 0.000} C_DIS
LIN {X 70.101,Y -41.986,Z -81.632,A -90.000,B 90.000,C 0.000} C_DIS
LIN {X 70.366,Y -41.946,Z -81.479,A -90.000,B 90.000,C 0.000} C_DIS
LIN {X 70.515,Y -41.917,Z -81.397,A -90.000,B 90.000,C 0.000} C_DIS
LIN {X 70.630,Y -41.884,Z -81.336,A -90.000,B 90.000,C 0.000} C_DIS
LIN {X 70.876,Y -41.810,Z -81.212,A -90.000,B 90.000,C 0.000} C_DIS
LIN {X 71.014,Y -41.769,Z -81.148,A -90.000,B 90.000,C 0.000} C_DIS
LIN {X 71.127,Y -41.730,Z -81.086,A -90.000,B 90.000,C 0.000} C_DIS
LIN {X 71.280,Y -41.688,Z -81.004,A -90.000,B 90.000,C 0.000} C_DIS
LIN {X 71.308,Y -41.679,Z -80.982,A -90.000,B 90.000,C 0.000} C_DIS
LIN {X 71.469,Y -41.619,Z -80.833,A -90.000,B 90.000,C 0.000} C_DIS
LIN {X 71.619,Y -41.565,Z -80.704,A -90.000,B 90.000,C 0.000} C_DIS
LIN {X 71.871,Y -41.476,Z -80.495,A -90.000,B 90.000,C 0.000} C_DIS
LIN {X 72.019,Y -41.414,Z -80.382,A -90.000,B 90.000,C 0.000} C_DIS
LIN {X 72.231,Y -41.308,Z -80.231,A -90.000,B 90.000,C 0.000} C_DIS
LIN {X 72.520,Y -41.159,Z -80.027,A -90.000,B 90.000,C 0.000} C_DIS
LIN {X 72.773,Y -41.017,Z -79.853,A -90.000,B 90.000,C 0.000} C_DIS
LIN {X 72.992,Y -40.908,Z -79.707,A -90.000,B 90.000,C 0.000} C_DIS
LIN {X 73.258,Y -40.781,Z -79.539,A -90.000,B 90.000,C 0.000} C_DIS
LIN {X 73.395,Y -40.711,Z -79.461,A -90.000,B 90.000,C 0.000} C_DIS
LIN {X 73.452,Y -40.682,Z -79.431,A -90.000,B 90.000,C 0.000} C_DIS
LIN {X 73.543,Y -40.635,Z -79.389,A -90.000,B 90.000,C 0.000} C_DIS
LIN {X 73.606,Y -40.605,Z -79.371,A -90.000,B 90.000,C 0.000} C_DIS
LIN {X 73.627,Y -40.597,Z -79.370,A -90.000,B 90.000,C 0.000} C_DIS
LIN {X 73.634,Y -40.595,Z -79.372,A -90.000,B 90.000,C 0.000} C_DIS
LIN {X 73.645,Y -40.594,Z -79.379,A -90.000,B 90.000,C 0.000} C_DIS
LIN {X 73.648,Y -40.598,Z -79.392,A -90.000,B 90.000,C 0.000} C_DIS
LIN {X 73.642,Y -40.612,Z -79.421,A -90.000,B 90.000,C 0.000} C_DIS
LIN {X 73.630,Y -40.626,Z -79.447,A -90.000,B 90.000,C 0.000} C_DIS
LIN {X 73.587,Y -40.668,Z -79.512,A -90.000,B 90.000,C 0.000} C_DIS
LIN {X 73.479,Y -40.755,Z -79.645,A -90.000,B 90.000,C 0.000} C_DIS
LIN {X 73.321,Y -40.865,Z -79.815,A -90.000,B 90.000,C 0.000} C_DIS
LIN {X 73.191,Y -40.947,Z -79.948,A -90.000,B 90.000,C 0.000} C_DIS
LIN {X 72.873,Y -41.137,Z -80.256,A -90.000,B 90.000,C 0.000} C_DIS
LIN {X 72.488,Y -41.363,Z -80.613,A -90.000,B 90.000,C 0.000} C_DIS
LIN {X 72.272,Y -41.484,Z -80.807,A -90.000,B 90.000,C 0.000} C_DIS
LIN {X 72.043,Y -41.593,Z -81.011,A -90.000,B 90.000,C 0.000} C_DIS
LIN {X 71.801,Y -41.685,Z -81.222,A -90.000,B 90.000,C 0.000} C_DIS
LIN {X 71.284,Y -41.863,Z -81.666,A -90.000,B 90.000,C 0.000} C_DIS
LIN {X 71.012,Y -41.956,Z -81.897,A -90.000,B 90.000,C 0.000} C_DIS
LIN {X 70.730,Y -42.045,Z -82.131,A -90.000,B 90.000,C 0.000} C_DIS
LIN {X 70.442,Y -42.109,Z -82.368,A -90.000,B 90.000,C 0.000} C_DIS
LIN {X 69.849,Y -42.181,Z -82.849,A -90.000,B 90.000,C 0.000} C_DIS
LIN {X 69.241,Y -42.254,Z -83.329,A -90.000,B 90.000,C 0.000} C_DIS
LIN {X 68.933,Y -42.273,Z -83.567,A -90.000,B 90.000,C 0.000} C_DIS
LIN {X 68.626,Y -42.261,Z -83.802,A -90.000,B 90.000,C 0.000} C_DIS
LIN {X 68.319,Y -42.228,Z -84.033,A -90.000,B 90.000,C 0.000} C_DIS
LIN {X 67.711,Y -42.158,Z -84.478,A -90.000,B 90.000,C 0.000} C_DIS
LIN {X 67.412,Y -42.125,Z -84.691,A -90.000,B 90.000,C 0.000} C_DIS
LIN {X 67.119,Y -42.081,Z -84.896,A -90.000,B 90.000,C 0.000} C_DIS
LIN {X 66.974,Y -42.049,Z -84.995,A -90.000,B 90.000,C 0.000} C_DIS
LIN {X 66.831,Y -42.012,Z -85.091,A -90.000,B 90.000,C 0.000} C_DIS
LIN {X 66.551,Y -41.937,Z -85.277,A -90.000,B 90.000,C 0.000} C_DIS
LIN {X 66.279,Y -41.865,Z -85.451,A -90.000,B 90.000,C 0.000} C_DIS
LIN {X 65.888,Y -41.755,Z -85.689,A -90.000,B 90.000,C 0.000} C_DIS
LIN {X 65.523,Y -41.651,Z -85.897,A -90.000,B 90.000,C 0.000} C_DIS
LIN {X 65.407,Y -41.614,Z -85.958,A -90.000,B 90.000,C 0.000} C_DIS
LIN {X 65.295,Y -41.575,Z -86.016,A -90.000,B 90.000,C 0.000} C_DIS
LIN {X 65.186,Y -41.533,Z -86.070,A -90.000,B 90.000,C 0.000} C_DIS
LIN {X 64.980,Y -41.449,Z -86.165,A -90.000,B 90.000,C 0.000} C_DIS
LIN {X 64.882,Y -41.411,Z -86.206,A -90.000,B 90.000,C 0.000} C_DIS
LIN {X 64.699,Y -41.340,Z -86.274,A -90.000,B 90.000,C 0.000} C_DIS
LIN {X 64.613,Y -41.307,Z -86.300,A -90.000,B 90.000,C 0.000} C_DIS
LIN {X 64.456,Y -41.245,Z -86.339,A -90.000,B 90.000,C 0.000} C_DIS
LIN {X 64.350,Y -41.204,Z -86.354,A -90.000,B 90.000,C 0.000} C_DIS
LIN {X 64.286,Y -41.179,Z -86.358,A -90.000,B 90.000,C 0.000} C_DIS
LIN {X 64.199,Y -41.144,Z -86.353,A -90.000,B 90.000,C 0.000} C_DIS
LIN {X 64.147,Y -41.123,Z -86.342,A -90.000,B 90.000,C 0.000} C_DIS
LIN {X 64.080,Y -41.096,Z -86.315,A -90.000,B 90.000,C 0.000} C_DIS
LIN {X 64.042,Y -41.081,Z -86.290,A -90.000,B 90.000,C 0.000} C_DIS
LIN {X 64.010,Y -41.068,Z -86.258,A -90.000,B 90.000,C 0.000} C_DIS
LIN {X 63.996,Y -41.062,Z -86.240,A -90.000,B 90.000,C 0.000} C_DIS
LIN {X 63.973,Y -41.052,Z -86.199,A -90.000,B 90.000,C 0.000} C_DIS
LIN {X 63.956,Y -41.044,Z -86.152,A -90.000,B 90.000,C 0.000} C_DIS
LIN {X 63.949,Y -41.041,Z -86.126,A -90.000,B 90.000,C 0.000} C_DIS
LIN {X 63.941,Y -41.037,Z -86.068,A -90.000,B 90.000,C 0.000} C_DIS
LIN {X 63.940,Y -41.035,Z -86.004,A -90.000,B 90.000,C 0.000} C_DIS
LIN {X 63.945,Y -41.035,Z -85.933,A -90.000,B 90.000,C 0.000} C_DIS
LIN {X 63.956,Y -41.039,Z -85.855,A -90.000,B 90.000,C 0.000} C_DIS
LIN {X 63.975,Y -41.047,Z -85.769,A -90.000,B 90.000,C 0.000} C_DIS
LIN {X 64.000,Y -41.058,Z -85.677,A -90.000,B 90.000,C 0.000} C_DIS
LIN {X 64.033,Y -41.072,Z -85.577,A -90.000,B 90.000,C 0.000} C_DIS
LIN {X 64.095,Y -41.099,Z -85.412,A -90.000,B 90.000,C 0.000} C_DIS
LIN {X 64.146,Y -41.120,Z -85.293,A -90.000,B 90.000,C 0.000} C_DIS
LIN {X 64.271,Y -41.172,Z -85.031,A -90.000,B 90.000,C 0.000} C_DIS
LIN {X 64.427,Y -41.240,Z -84.737,A -90.000,B 90.000,C 0.000} C_DIS
LIN {X 64.517,Y -41.275,Z -84.577,A -90.000,B 90.000,C 0.000} C_DIS
LIN {X 64.615,Y -41.308,Z -84.408,A -90.000,B 90.000,C 0.000} C_DIS
LIN {X 64.659,Y -41.323,Z -84.334,A -90.000,B 90.000,C 0.000} C_DIS
LIN {X 64.769,Y -41.350,Z -84.155,A -90.000,B 90.000,C 0.000} C_DIS
LIN {X 64.834,Y -41.368,Z -84.057,A -90.000,B 90.000,C 0.000} C_DIS
LIN {X 65.180,Y -41.477,Z -83.545,A -90.000,B 90.000,C 0.000} C_DIS
LIN {X 65.280,Y -41.508,Z -83.399,A -90.000,B 90.000,C 0.000} C_DIS
LIN {X 65.505,Y -41.579,Z -83.092,A -90.000,B 90.000,C 0.000} C_DIS
LIN {X 65.690,Y -41.633,Z -82.855,A -90.000,B 90.000,C 0.000} C_DIS
LIN {X 65.881,Y -41.690,Z -82.628,A -90.000,B 90.000,C 0.000} C_DIS
LIN {X 65.970,Y -41.710,Z -82.529,A -90.000,B 90.000,C 0.000} C_DIS
LIN {X 66.113,Y -41.728,Z -82.378,A -90.000,B 90.000,C 0.000} C_DIS
LIN {X 66.394,Y -41.764,Z -82.086,A -90.000,B 90.000,C 0.000} C_DIS
LIN {X 66.658,Y -41.796,Z -81.831,A -90.000,B 90.000,C 0.000} C_DIS
LIN {X 67.000,Y -41.838,Z -81.521,A -90.000,B 90.000,C 0.000} C_DIS
LIN {X 67.151,Y -41.857,Z -81.390,A -90.000,B 90.000,C 0.000} C_DIS
LIN {X 67.356,Y -41.883,Z -81.219,A -90.000,B 90.000,C 0.000} C_DIS
LIN {X 67.476,Y -41.896,Z -81.111,A -90.000,B 90.000,C 0.000} C_DIS
LIN {X 67.576,Y -41.902,Z -81.023,A -90.000,B 90.000,C 0.000} C_DIS
LIN {X 67.694,Y -41.904,Z -80.921,A -90.000,B 90.000,C 0.000} C_DIS
LIN {X 67.838,Y -41.899,Z -80.799,A -90.000,B 90.000,C 0.000} C_DIS
LIN {X 67.958,Y -41.891,Z -80.702,A -90.000,B 90.000,C 0.000} C_DIS
LIN {X 68.111,Y -41.875,Z -80.585,A -90.000,B 90.000,C 0.000} C_DIS
LIN {X 68.226,Y -41.855,Z -80.500,A -90.000,B 90.000,C 0.000} C_DIS
LIN {X 68.562,Y -41.788,Z -80.266,A -90.000,B 90.000,C 0.000} C_DIS
LIN {X 68.600,Y -41.779,Z -80.240,A -90.000,B 90.000,C 0.000} C_DIS
LIN {X 69.010,Y -41.719,Z -79.977,A -90.000,B 90.000,C 0.000} C_DIS
LIN {X 69.149,Y -41.700,Z -79.895,A -90.000,B 90.000,C 0.000} C_DIS
LIN {X 69.473,Y -41.657,Z -79.709,A -90.000,B 90.000,C 0.000} C_DIS
LIN {X 69.651,Y -41.630,Z -79.611,A -90.000,B 90.000,C 0.000} C_DIS
LIN {X 69.806,Y -41.597,Z -79.530,A -90.000,B 90.000,C 0.000} C_DIS
LIN {X 69.978,Y -41.547,Z -79.445,A -90.000,B 90.000,C 0.000} C_DIS
LIN {X 70.054,Y -41.525,Z -79.409,A -90.000,B 90.000,C 0.000} C_DIS
LIN {X 70.090,Y -41.514,Z -79.389,A -90.000,B 90.000,C 0.000} C_DIS
LIN {X 70.249,Y -41.453,Z -79.250,A -90.000,B 90.000,C 0.000} C_DIS
LIN {X 70.530,Y -41.308,Z -79.020,A -90.000,B 90.000,C 0.000} C_DIS
LIN {X 70.729,Y -41.212,Z -78.855,A -90.000,B 90.000,C 0.000} C_DIS
LIN {X 70.901,Y -41.133,Z -78.711,A -90.000,B 90.000,C 0.000} C_DIS
LIN {X 71.047,Y -41.065,Z -78.586,A -90.000,B 90.000,C 0.000} C_DIS
LIN {X 71.263,Y -40.963,Z -78.392,A -90.000,B 90.000,C 0.000} C_DIS
LIN {X 71.335,Y -40.926,Z -78.321,A -90.000,B 90.000,C 0.000} C_DIS
LIN {X 71.384,Y -40.899,Z -78.268,A -90.000,B 90.000,C 0.000} C_DIS
LIN {X 71.411,Y -40.881,Z -78.230,A -90.000,B 90.000,C 0.000} C_DIS
LIN {X 71.416,Y -40.875,Z -78.217,A -90.000,B 90.000,C 0.000} C_DIS
LIN {X 71.414,Y -40.872,Z -78.205,A -90.000,B 90.000,C 0.000} C_DIS
LIN {X 71.407,Y -40.872,Z -78.201,A -90.000,B 90.000,C 0.000} C_DIS
LIN {X 71.387,Y -40.877,Z -78.202,A -90.000,B 90.000,C 0.000} C_DIS
LIN {X 71.315,Y -40.900,Z -78.227,A -90.000,B 90.000,C 0.000} C_DIS
LIN {X 71.245,Y -40.924,Z -78.260,A -90.000,B 90.000,C 0.000} C_DIS
LIN {X 71.055,Y -40.992,Z -78.361,A -90.000,B 90.000,C 0.000} C_DIS
LIN {X 70.937,Y -41.035,Z -78.428,A -90.000,B 90.000,C 0.000} C_DIS
LIN {X 70.805,Y -41.090,Z -78.506,A -90.000,B 90.000,C 0.000} C_DIS
LIN {X 70.332,Y -41.306,Z -78.791,A -90.000,B 90.000,C 0.000} C_DIS
LIN {X 69.961,Y -41.453,Z -79.019,A -90.000,B 90.000,C 0.000} C_DIS
LIN {X 69.555,Y -41.565,Z -79.272,A -90.000,B 90.000,C 0.000} C_DIS
LIN {X 69.119,Y -41.637,Z -79.543,A -90.000,B 90.000,C 0.000} C_DIS
LIN {X 68.661,Y -41.703,Z -79.828,A -90.000,B 90.000,C 0.000} C_DIS
LIN {X 68.189,Y -41.800,Z -80.121,A -90.000,B 90.000,C 0.000} C_DIS
LIN {X 67.708,Y -41.850,Z -80.417,A -90.000,B 90.000,C 0.000} C_DIS
LIN {X 67.226,Y -41.833,Z -80.710,A -90.000,B 90.000,C 0.000} C_DIS
LIN {X 66.986,Y -41.802,Z -80.854,A -90.000,B 90.000,C 0.000} C_DIS
LIN {X 66.286,Y -41.705,Z -81.267,A -90.000,B 90.000,C 0.000} C_DIS
LIN {X 65.841,Y -41.642,Z -81.521,A -90.000,B 90.000,C 0.000} C_DIS
LIN {X 65.629,Y -41.608,Z -81.639,A -90.000,B 90.000,C 0.000} C_DIS
LIN {X 65.424,Y -41.562,Z -81.750,A -90.000,B 90.000,C 0.000} C_DIS
LIN {X 65.227,Y -41.507,Z -81.854,A -90.000,B 90.000,C 0.000} C_DIS
LIN {X 64.863,Y -41.387,Z -82.038,A -90.000,B 90.000,C 0.000} C_DIS
LIN {X 64.618,Y -41.306,Z -82.151,A -90.000,B 90.000,C 0.000} C_DIS
LIN {X 64.400,Y -41.234,Z -82.241,A -90.000,B 90.000,C 0.000} C_DIS
LIN {X 64.214,Y -41.174,Z -82.305,A -90.000,B 90.000,C 0.000} C_DIS
LIN {X 64.107,Y -41.140,Z -82.333,A -90.000,B 90.000,C 0.000} C_DIS
LIN {X 64.017,Y -41.112,Z -82.347,A -90.000,B 90.000,C 0.000} C_DIS
LIN {X 63.978,Y -41.100,Z -82.349,A -90.000,B 90.000,C 0.000} C_DIS
LIN {X 63.928,Y -41.084,Z -82.346,A -90.000,B 90.000,C 0.000} C_DIS
LIN {X 63.900,Y -41.075,Z -82.339,A -90.000,B 90.000,C 0.000} C_DIS
LIN {X 63.876,Y -41.067,Z -82.329,A -90.000,B 90.000,C 0.000} C_DIS
LIN {X 63.857,Y -41.061,Z -82.314,A -90.000,B 90.000,C 0.000} C_DIS
LIN {X 63.843,Y -41.057,Z -82.296,A -90.000,B 90.000,C 0.000} C_DIS
LIN {X 63.834,Y -41.054,Z -82.274,A -90.000,B 90.000,C 0.000} C_DIS
LIN {X 63.829,Y -41.053,Z -82.248,A -90.000,B 90.000,C 0.000} C_DIS
LIN {X 63.830,Y -41.053,Z -82.218,A -90.000,B 90.000,C 0.000} C_DIS
LIN {X 63.841,Y -41.056,Z -82.164,A -90.000,B 90.000,C 0.000} C_DIS
LIN {X 63.874,Y -41.068,Z -82.078,A -90.000,B 90.000,C 0.000} C_DIS
LIN {X 63.930,Y -41.088,Z -81.973,A -90.000,B 90.000,C 0.000} C_DIS
LIN {X 64.009,Y -41.116,Z -81.850,A -90.000,B 90.000,C 0.000} C_DIS
LIN {X 64.111,Y -41.151,Z -81.707,A -90.000,B 90.000,C 0.000} C_DIS
LIN {X 64.312,Y -41.221,Z -81.455,A -90.000,B 90.000,C 0.000} C_DIS
LIN {X 64.572,Y -41.308,Z -81.156,A -90.000,B 90.000,C 0.000} C_DIS
LIN {X 64.694,Y -41.348,Z -81.020,A -90.000,B 90.000,C 0.000} C_DIS
LIN {X 64.957,Y -41.427,Z -80.736,A -90.000,B 90.000,C 0.000} C_DIS
LIN {X 65.054,Y -41.447,Z -80.636,A -90.000,B 90.000,C 0.000} C_DIS
LIN {X 65.353,Y -41.488,Z -80.346,A -90.000,B 90.000,C 0.000} C_DIS
LIN {X 65.696,Y -41.528,Z -80.037,A -90.000,B 90.000,C 0.000} C_DIS
LIN {X 65.913,Y -41.554,Z -79.849,A -90.000,B 90.000,C 0.000} C_DIS
LIN {X 66.081,Y -41.574,Z -79.709,A -90.000,B 90.000,C 0.000} C_DIS
LIN {X 66.345,Y -41.606,Z -79.473,A -90.000,B 90.000,C 0.000} C_DIS
LIN {X 66.619,Y -41.637,Z -79.234,A -90.000,B 90.000,C 0.000} C_DIS
LIN {X 66.737,Y -41.646,Z -79.138,A -90.000,B 90.000,C 0.000} C_DIS
LIN {X 66.874,Y -41.648,Z -79.029,A -90.000,B 90.000,C 0.000} C_DIS
LIN {X 67.018,Y -41.645,Z -78.920,A -90.000,B 90.000,C 0.000} C_DIS
LIN {X 67.169,Y -41.636,Z -78.811,A -90.000,B 90.000,C 0.000} C_DIS
LIN {X 67.291,Y -41.625,Z -78.724,A -90.000,B 90.000,C 0.000} C_DIS
LIN {X 67.399,Y -41.609,Z -78.649,A -90.000,B 90.000,C 0.000} C_DIS
LIN {X 67.505,Y -41.587,Z -78.578,A -90.000,B 90.000,C 0.000} C_DIS
LIN {X 67.751,Y -41.539,Z -78.421,A -90.000,B 90.000,C 0.000} C_DIS
LIN {X 67.839,Y -41.517,Z -78.366,A -90.000,B 90.000,C 0.000} C_DIS
LIN {X 67.972,Y -41.488,Z -78.283,A -90.000,B 90.000,C 0.000} C_DIS
LIN {X 68.141,Y -41.452,Z -78.185,A -90.000,B 90.000,C 0.000} C_DIS
LIN {X 68.486,Y -41.375,Z -77.993,A -90.000,B 90.000,C 0.000} C_DIS
LIN {X 68.717,Y -41.325,Z -77.869,A -90.000,B 90.000,C 0.000} C_DIS
LIN {X 68.794,Y -41.308,Z -77.829,A -90.000,B 90.000,C 0.000} C_DIS
LIN {X 68.794,Y -60.000,Z -77.829,A -90.000,B 90.000,C 0.000} C_DIS
LIN {X 56.246,Y -60.000,Z -70.848,A -90.000,B 90.000,C 0.000} C_DIS
LIN {X 56.246,Y -42.588,Z -70.848,A -90.000,B 90.000,C 0.000} C_DIS
LIN {X 56.168,Y -42.576,Z -70.985,A -90.000,B 90.000,C 0.000} C_DIS
LIN {X 56.029,Y -42.566,Z -71.217,A -90.000,B 90.000,C 0.000} C_DIS
LIN {X 55.956,Y -42.562,Z -71.332,A -90.000,B 90.000,C 0.000} C_DIS
LIN {X 55.922,Y -42.562,Z -71.379,A -90.000,B 90.000,C 0.000} C_DIS
LIN {X 55.840,Y -42.562,Z -71.485,A -90.000,B 90.000,C 0.000} C_DIS
LIN {X 55.654,Y -42.567,Z -71.708,A -90.000,B 90.000,C 0.000} C_DIS
LIN {X 55.584,Y -42.570,Z -71.789,A -90.000,B 90.000,C 0.000} C_DIS
LIN {X 55.324,Y -42.584,Z -72.070,A -90.000,B 90.000,C 0.000} C_DIS
LIN {X 55.270,Y -42.588,Z -72.124,A -90.000,B 90.000,C 0.000} C_DIS
LIN {X 55.136,Y -42.599,Z -72.248,A -90.000,B 90.000,C 0.000} C_DIS
LIN {X 54.880,Y -42.611,Z -72.505,A -90.000,B 90.000,C 0.000} C_DIS
LIN {X 54.687,Y -42.603,Z -72.690,A -90.000,B 90.000,C 0.000} C_DIS
LIN {X 54.583,Y -42.596,Z -72.788,A -90.000,B 90.000,C 0.000} C_DIS
LIN {X 54.425,Y -42.585,Z -72.938,A -90.000,B 90.000,C 0.000} C_DIS
LIN {X 54.228,Y -42.560,Z -73.117,A -90.000,B 90.000,C 0.000} C_DIS
LIN {X 53.913,Y -42.515,Z -73.398,A -90.000,B 90.000,C 0.000} C_DIS
LIN {X 53.628,Y -42.488,Z -73.621,A -90.000,B 90.000,C 0.000} C_DIS
LIN {X 53.549,Y -42.482,Z -73.679,A -90.000,B 90.000,C 0.000} C_DIS
LIN {X 53.146,Y -42.456,Z -73.963,A -90.000,B 90.000,C 0.000} C_DIS
LIN {X 53.027,Y -42.453,Z -74.036,A -90.000,B 90.000,C 0.000} C_DIS
LIN {X 52.742,Y -42.449,Z -74.201,A -90.000,B 90.000,C 0.000} C_DIS
LIN {X 52.626,Y -42.450,Z -74.263,A -90.000,B 90.000,C 0.000} C_DIS
LIN {X 52.396,Y -42.455,Z -74.377,A -90.000,B 90.000,C 0.000} C_DIS
LIN {X 52.213,Y -42.456,Z -74.466,A -90.000,B 90.000,C 0.000} C_DIS
LIN {X 51.951,Y -42.447,Z -74.587,A -90.000,B 90.000,C 0.000} C_DIS
LIN {X 51.790,Y -42.437,Z -74.660,A -90.000,B 90.000,C 0.000} C_DIS
LIN {X 51.660,Y -42.432,Z -74.714,A -90.000,B 90.000,C 0.000} C_DIS
LIN {X 51.362,Y -42.425,Z -74.827,A -90.000,B 90.000,C 0.000} C_DIS
LIN {X 51.244,Y -42.424,Z -74.868,A -90.000,B 90.000,C 0.000} C_DIS
LIN {X 50.734,Y -42.428,Z -75.029,A -90.000,B 90.000,C 0.000} C_DIS
LIN {X 49.485,Y -42.434,Z -75.422,A -90.000,B 90.000,C 0.000} C_DIS
LIN {X 49.206,Y -42.432,Z -75.513,A -90.000,B 90.000,C 0.000} C_DIS
LIN {X 48.868,Y -42.418,Z -75.617,A -90.000,B 90.000,C 0.000} C_DIS
LIN {X 48.754,Y -42.414,Z -75.646,A -90.000,B 90.000,C 0.000} C_DIS
LIN {X 48.423,Y -42.411,Z -75.716,A -90.000,B 90.000,C 0.000} C_DIS
LIN {X 48.330,Y -42.410,Z -75.734,A -90.000,B 90.000,C 0.000} C_DIS
LIN {X 48.207,Y -42.412,Z -75.754,A -90.000,B 90.000,C 0.000} C_DIS
LIN {X 48.022,Y -42.418,Z -75.777,A -90.000,B 90.000,C 0.000} C_DIS
LIN {X 47.794,Y -42.429,Z -75.796,A -90.000,B 90.000,C 0.000} C_DIS
LIN {X 47.658,Y -42.437,Z -75.803,A -90.000,B 90.000,C 0.000} C_DIS
LIN {X 47.507,Y -42.449,Z -75.805,A -90.000,B 90.000,C 0.000} C_DIS
LIN {X 46.770,Y -42.515,Z -75.794,A -90.000,B 90.000,C 0.000} C_DIS
LIN {X 46.493,Y -42.527,Z -75.784,A -90.000,B 90.000,C 0.000} C_DIS
LIN {X 46.003,Y -42.531,Z -75.758,A -90.000,B 90.000,C 0.000} C_DIS
LIN {X 45.832,Y -42.531,Z -75.747,A -90.000,B 90.000,C 0.000} C_DIS
LIN {X 45.360,Y -42.537,Z -75.703,A -90.000,B 90.000,C 0.000} C_DIS
LIN {X 45.239,Y -42.541,Z -75.685,A -90.000,B 90.000,C 0.000} C_DIS
LIN {X 44.924,Y -42.555,Z -75.629,A -90.000,B 90.000,C 0.000} C_DIS
LIN {X 44.801,Y -42.562,Z -75.601,A -90.000,B 90.000,C 0.000} C_DIS
LIN {X 44.431,Y -42.589,Z -75.494,A -90.000,B 90.000,C 0.000} C_DIS
LIN {X 44.192,Y -42.599,Z -75.422,A -90.000,B 90.000,C 0.000} C_DIS
LIN {X 43.614,Y -42.604,Z -75.238,A -90.000,B 90.000,C 0.000} C_DIS
LIN {X 43.463,Y -42.603,Z -75.194,A -90.000,B 90.000,C 0.000} C_DIS
LIN {X 43.305,Y -42.605,Z -75.142,A -90.000,B 90.000,C 0.000} C_DIS
LIN {X 43.113,Y -42.611,Z -75.069,A -90.000,B 90.000,C 0.000} C_DIS
LIN {X 42.940,Y -42.617,Z -75.000,A -90.000,B 90.000,C 0.000} C_DIS
LIN {X 42.223,Y -42.625,Z -74.695,A -90.000,B 90.000,C 0.000} C_DIS
LIN {X 41.595,Y -42.479,Z -74.888,A -90.000,B 90.000,C 0.000} C_DIS
LIN {X 41.135,Y -42.387,Z -75.030,A -90.000,B 90.000,C 0.000} C_DIS
LIN {X 40.886,Y -42.340,Z -75.101,A -90.000,B 90.000,C 0.000} C_DIS
LIN {X 40.610,Y -42.289,Z -75.175,A -90.000,B 90.000,C 0.000} C_DIS
LIN {X 40.462,Y -42.274,Z -75.221,A -90.000,B 90.000,C 0.000} C_DIS
LIN {X 40.162,Y -42.249,Z -75.301,A -90.000,B 90.000,C 0.000} C_DIS
LIN {X 40.020,Y -42.239,Z -75.331,A -90.000,B 90.000,C 0.000} C_DIS
LIN {X 39.896,Y -42.228,Z -75.363,A -90.000,B 90.000,C 0.000} C_DIS
LIN {X 39.490,Y -42.214,Z -75.479,A -90.000,B 90.000,C 0.000} C_DIS
LIN {X 39.205,Y -42.208,Z -75.547,A -90.000,B 90.000,C 0.000} C_DIS
LIN {X 39.030,Y -42.197,Z -75.580,A -90.000,B 90.000,C 0.000} C_DIS
LIN {X 38.580,Y -42.209,Z -75.673,A -90.000,B 90.000,C 0.000} C_DIS
LIN {X 38.236,Y -42.210,Z -75.740,A -90.000,B 90.000,C 0.000} C_DIS
LIN {X 38.145,Y -42.206,Z -75.754,A -90.000,B 90.000,C 0.000} C_DIS
LIN {X 37.955,Y -42.204,Z -75.776,A -90.000,B 90.000,C 0.000} C_DIS
LIN {X 37.758,Y -42.208,Z -75.789,A -90.000,B 90.000,C 0.000} C_DIS
LIN {X 37.509,Y -42.223,Z -75.811,A -90.000,B 90.000,C 0.000} C_DIS
LIN {X 37.323,Y -42.235,Z -75.826,A -90.000,B 90.000,C 0.000} C_DIS
LIN {X 37.186,Y -42.236,Z -75.831,A -90.000,B 90.000,C 0.000} C_DIS
LIN {X 37.059,Y -42.236,Z -75.838,A -90.000,B 90.000,C 0.000} C_DIS
LIN {X 36.649,Y -42.234,Z -75.860,A -90.000,B 90.000,C 0.000} C_DIS
LIN {X 36.506,Y -42.235,Z -75.864,A -90.000,B 90.000,C 0.000} C_DIS
LIN {X 36.371,Y -42.242,Z -75.860,A -90.000,B 90.000,C 0.000} C_DIS
LIN {X 36.033,Y -42.244,Z -75.831,A -90.000,B 90.000,C 0.000} C_DIS
LIN {X 35.910,Y -42.247,Z -75.817,A -90.000,B 90.000,C 0.000} C_DIS
LIN {X 35.720,Y -42.255,Z -75.789,A -90.000,B 90.000,C 0.000} C_DIS
LIN {X 35.523,Y -42.271,Z -75.765,A -90.000,B 90.000,C 0.000} C_DIS
LIN {X 35.186,Y -42.284,Z -75.714,A -90.000,B 90.000,C 0.000} C_DIS
LIN {X 35.108,Y -42.281,Z -75.700,A -90.000,B 90.000,C 0.000} C_DIS
LIN {X 34.975,Y -42.280,Z -75.670,A -90.000,B 90.000,C 0.000} C_DIS
LIN {X 34.672,Y -42.278,Z -75.598,A -90.000,B 90.000,C 0.000} C_DIS
LIN {X 34.549,Y -42.279,Z -75.564,A -90.000,B 90.000,C 0.000} C_DIS
LIN {X 34.494,Y -42.280,Z -75.547,A -90.000,B 90.000,C 0.000} C_DIS
LIN {X 34.364,Y -42.285,Z -75.506,A -90.000,B 90.000,C 0.000} C_DIS
LIN {X 34.151,Y -42.301,Z -75.430,A -90.000,B 90.000,C 0.000} C_DIS
LIN {X 33.986,Y -42.303,Z -75.360,A -90.000,B 90.000,C 0.000} C_DIS
LIN {X 33.830,Y -42.309,Z -75.289,A -90.000,B 90.000,C 0.000} C_DIS
LIN {X 33.360,Y -42.298,Z -75.046,A -90.000,B 90.000,C 0.000} C_DIS
LIN {X 33.283,Y -42.298,Z -75.006,A -90.000,B 90.000,C 0.000} C_DIS
LIN {X 33.089,Y -42.298,Z -74.896,A -90.000,B 90.000,C 0.000} C_DIS
LIN {X 32.979,Y -42.300,Z -74.830,A -90.000,B 90.000,C 0.000} C_DIS
LIN {X 32.942,Y -42.298,Z -74.805,A -90.000,B 90.000,C 0.000} C_DIS
LIN {X 32.800,Y -42.293,Z -74.706,A -90.000,B 90.000,C 0.000} C_DIS
LIN {X 32.695,Y -42.293,Z -74.625,A -90.000,B 90.000,C 0.000} C_DIS
LIN {X 32.605,Y -42.285,Z -74.550,A -90.000,B 90.000,C 0.000} C_DIS
LIN {X 32.436,Y -42.275,Z -74.399,A -90.000,B 90.000,C 0.000} C_DIS
LIN {X 32.349,Y -42.266,Z -74.308,A -90.000,B 90.000,C 0.000} C_DIS
LIN {X 32.150,Y -42.248,Z -74.086,A -90.000,B 90.000,C 0.000} C_DIS
LIN {X 32.030,Y -42.238,Z -73.946,A -90.000,B 90.000,C 0.000} C_DIS
LIN {X 31.853,Y -42.229,Z -73.724,A -90.000,B 90.000,C 0.000} C_DIS
LIN {X 31.735,Y -42.216,Z -73.568,A -90.000,B 90.000,C 0.000} C_DIS
LIN {X 31.689,Y -42.208,Z -73.504,A -90.000,B 90.000,C 0.000} C_DIS
LIN {X 31.613,Y -42.197,Z -73.394,A -90.000,B 90.000,C 0.000} C_DIS
LIN {X 31.534,Y -42.187,Z -73.275,A -90.000,B 90.000,C 0.000} C_DIS
LIN {X 31.430,Y -42.159,Z -73.097,A -90.000,B 90.000,C 0.000} C_DIS
LIN {X 31.368,Y -42.144,Z -72.983,A -90.000,B 90.000,C 0.000} C_DIS
LIN {X 31.331,Y -42.132,Z -72.900,A -90.000,B 90.000,C 0.000} C_DIS
LIN {X 31.194,Y -42.091,Z -72.575,A -90.000,B 90.000,C 0.000} C_DIS
LIN {X 31.153,Y -42.080,Z -72.471,A -90.000,B 90.000,C 0.000} C_DIS
LIN {X 31.056,Y -42.034,Z -72.141,A -90.000,B 90.000,C 0.000} C_DIS
LIN {X 31.052,Y -42.031,Z -72.125,A -90.000,B 90.000,C 0.000} C_DIS
LIN {X 30.967,Y -41.978,Z -71.764,A -90.000,B 90.000,C 0.000} C_DIS
LIN {X 30.949,Y -41.970,Z -71.695,A -90.000,B 90.000,C 0.000} C_DIS
LIN {X 30.913,Y -41.959,Z -71.546,A -90.000,B 90.000,C 0.000} C_DIS
LIN {X 30.905,Y -41.957,Z -71.504,A -90.000,B 90.000,C 0.000} C_DIS
LIN {X 30.836,Y -41.932,Z -71.086,A -90.000,B 90.000,C 0.000} C_DIS
LIN {X 30.808,Y -41.904,Z -70.809,A -90.000,B 90.000,C 0.000} C_DIS
LIN {X 30.784,Y -41.879,Z -70.586,A -90.000,B 90.000,C 0.000} C_DIS
LIN {X 30.754,Y -41.827,Z -70.197,A -90.000,B 90.000,C 0.000} C_DIS
LIN {X 30.752,Y -41.802,Z -70.032,A -90.000,B 90.000,C 0.000} C_DIS
LIN {X 30.757,Y -41.762,Z -69.740,A -90.000,B 90.000,C 0.000} C_DIS
LIN {X 30.762,Y -41.742,Z -69.592,A -90.000,B 90.000,C 0.000} C_DIS
LIN {X 30.777,Y -41.716,Z -69.343,A -90.000,B 90.000,C 0.000} C_DIS
LIN {X 30.800,Y -41.693,Z -69.065,A -90.000,B 90.000,C 0.000} C_DIS
LIN {X 30.801,Y -41.691,Z -69.023,A -90.000,B 90.000,C 0.000} C_DIS
LIN {X 30.811,Y -41.684,Z -68.915,A -90.000,B 90.000,C 0.000} C_DIS
LIN {X 30.887,Y -41.646,Z -68.112,A -90.000,B 90.000,C 0.000} C_DIS
LIN {X 30.906,Y -41.642,Z -67.934,A -90.000,B 90.000,C 0.000} C_DIS
LIN {X 30.931,Y -41.634,Z -67.783,A -90.000,B 90.000,C 0.000} C_DIS
LIN {X 30.960,Y -41.624,Z -67.622,A -90.000,B 90.000,C 0.000} C_DIS
LIN {X 30.956,Y -41.636,Z -67.295,A -90.000,B 90.000,C 0.000} C_DIS
LIN {X 30.956,Y -41.647,Z -66.970,A -90.000,B 90.000,C 0.000} C_DIS
LIN {X 31.008,Y -41.653,Z -66.504,A -90.000,B 90.000,C 0.000} C_DIS
LIN {X 31.027,Y -41.656,Z -66.366,A -90.000,B 90.000,C 0.000} C_DIS
LIN {X 31.205,Y -41.670,Z -65.287,A -90.000,B 90.000,C 0.000} C_DIS
LIN {X 31.233,Y -41.668,Z -65.146,A -90.000,B 90.000,C 0.000} C_DIS
LIN {X 31.270,Y -41.668,Z -64.995,A -90.000,B 90.000,C 0.000} C_DIS
LIN {X 31.338,Y -41.660,Z -64.771,A -90.000,B 90.000,C 0.000} C_DIS
LIN {X 31.486,Y -41.644,Z -64.304,A -90.000,B 90.000,C 0.000} C_DIS
LIN {X 31.571,Y -41.628,Z -64.077,A -90.000,B 90.000,C 0.000} C_DIS
LIN {X 31.703,Y -41.604,Z -63.737,A -90.000,B 90.000,C 0.000} C_DIS
LIN {X 31.799,Y -41.615,Z -63.305,A -90.000,B 90.000,C 0.000} C_DIS
LIN {X 31.910,Y -41.630,Z -62.882,A -90.000,B 90.000,C 0.000} C_DIS
LIN {X 32.187,Y -41.691,Z -61.884,A -90.000,B 90.000,C 0.000} C_DIS
LIN {X 32.369,Y -41.711,Z -61.323,A -90.000,B 90.000,C 0.000} C_DIS
LIN {X 32.508,Y -41.740,Z -60.926,A -90.000,B 90.000,C 0.000} C_DIS
LIN {X 32.705,Y -41.777,Z -60.386,A -90.000,B 90.000,C 0.000} C_DIS
LIN {X 32.922,Y -41.814,Z -59.807,A -90.000,B 90.000,C 0.000} C_DIS
LIN {X 33.003,Y -41.822,Z -59.610,A -90.000,B 90.000,C 0.000} C_DIS
LIN {X 33.080,Y -41.833,Z -59.431,A -90.000,B 90.000,C 0.000} C_DIS
LIN {X 33.190,Y -41.846,Z -59.185,A -90.000,B 90.000,C 0.000} C_DIS
LIN {X 33.238,Y -41.854,Z -59.084,A -90.000,B 90.000,C 0.000} C_DIS
LIN {X 33.351,Y -41.882,Z -58.863,A -90.000,B 90.000,C 0.000} C_DIS
LIN {X 33.677,Y -41.925,Z -58.309,A -90.000,B 90.000,C 0.000} C_DIS
LIN {X 33.763,Y -41.939,Z -58.168,A -90.000,B 90.000,C 0.000} C_DIS
LIN {X 34.061,Y -41.982,Z -57.690,A -90.000,B 90.000,C 0.000} C_DIS
LIN {X 34.291,Y -42.005,Z -57.335,A -90.000,B 90.000,C 0.000} C_DIS
LIN {X 34.339,Y -42.006,Z -57.268,A -90.000,B 90.000,C 0.000} C_DIS
LIN {X 34.520,Y -42.021,Z -57.030,A -90.000,B 90.000,C 0.000} C_DIS
LIN {X 34.615,Y -42.023,Z -56.915,A -90.000,B 90.000,C 0.000} C_DIS
LIN {X 34.703,Y -42.026,Z -56.813,A -90.000,B 90.000,C 0.000} C_DIS
LIN {X 34.835,Y -42.036,Z -56.667,A -90.000,B 90.000,C 0.000} C_DIS
LIN {X 35.130,Y -42.063,Z -56.336,A -90.000,B 90.000,C 0.000} C_DIS
LIN {X 35.569,Y -42.104,Z -55.897,A -90.000,B 90.000,C 0.000} C_DIS
LIN {X 35.613,Y -42.104,Z -55.858,A -90.000,B 90.000,C 0.000} C_DIS
LIN {X 35.715,Y -42.105,Z -55.766,A -90.000,B 90.000,C 0.000} C_DIS
LIN {X 35.844,Y -42.106,Z -55.651,A -90.000,B 90.000,C 0.000} C_DIS
LIN {X 35.946,Y -42.111,Z -55.569,A -90.000,B 90.000,C 0.000} C_DIS
LIN {X 36.166,Y -42.128,Z -55.401,A -90.000,B 90.000,C 0.000} C_DIS
LIN {X 36.318,Y -42.141,Z -55.287,A -90.000,B 90.000,C 0.000} C_DIS
LIN {X 36.404,Y -42.151,Z -55.227,A -90.000,B 90.000,C 0.000} C_DIS
LIN {X 36.567,Y -42.170,Z -55.120,A -90.000,B 90.000,C 0.000} C_DIS
LIN {X 36.896,Y -42.190,Z -54.920,A -90.000,B 90.000,C 0.000} C_DIS
LIN {X 37.129,Y -42.186,Z -54.795,A -90.000,B 90.000,C 0.000} C_DIS
LIN {X 37.647,Y -42.177,Z -54.522,A -90.000,B 90.000,C 0.000} C_DIS
LIN {X 37.860,Y -42.182,Z -54.424,A -90.000,B 90.000,C 0.000} C_DIS
LIN {X 38.049,Y -42.193,Z -54.347,A -90.000,B 90.000,C 0.000} C_DIS
LIN {X 38.188,Y -42.192,Z -54.297,A -90.000,B 90.000,C 0.000} C_DIS
LIN {X 38.360,Y -42.196,Z -54.242,A -90.000,B 90.000,C 0.000} C_DIS
LIN {X 38.408,Y -42.199,Z -54.229,A -90.000,B 90.000,C 0.000} C_DIS
LIN {X 38.779,Y -42.199,Z -54.150,A -90.000,B 90.000,C 0.000} C_DIS
LIN {X 39.558,Y -42.192,Z -53.994,A -90.000,B 90.000,C 0.000} C_DIS
LIN {X 39.719,Y -42.189,Z -53.964,A -90.000,B 90.000,C 0.000} C_DIS
LIN {X 39.894,Y -42.182,Z -53.942,A -90.000,B 90.000,C 0.000} C_DIS
LIN {X 40.082,Y -42.183,Z -53.929,A -90.000,B 90.000,C 0.000} C_DIS
LIN {X 40.363,Y -42.167,Z -53.923,A -90.000,B 90.000,C 0.000} C_DIS
LIN {X 40.453,Y -42.164,Z -53.925,A -90.000,B 90.000,C 0.000} C_DIS
LIN {X 40.877,Y -42.154,Z -53.964,A -90.000,B 90.000,C 0.000} C_DIS
LIN {X 41.002,Y -42.154,Z -53.978,A -90.000,B 90.000,C 0.000} C_DIS
LIN {X 41.502,Y -42.164,Z -54.049,A -90.000,B 90.000,C 0.000} C_DIS
LIN {X 41.732,Y -42.164,Z -54.085,A -90.000,B 90.000,C 0.000} C_DIS
LIN {X 41.912,Y -42.161,Z -54.115,A -90.000,B 90.000,C 0.000} C_DIS
LIN {X 42.129,Y -42.149,Z -54.160,A -90.000,B 90.000,C 0.000} C_DIS
LIN {X 42.286,Y -42.139,Z -54.198,A -90.000,B 90.000,C 0.000} C_DIS
LIN {X 42.519,Y -42.113,Z -54.262,A -90.000,B 90.000,C 0.000} C_DIS
LIN {X 42.646,Y -42.099,Z -54.304,A -90.000,B 90.000,C 0.000} C_DIS
LIN {X 42.857,Y -42.080,Z -54.387,A -90.000,B 90.000,C 0.000} C_DIS
LIN {X 43.130,Y -42.058,Z -54.497,A -90.000,B 90.000,C 0.000} C_DIS
LIN {X 43.249,Y -42.053,Z -54.553,A -90.000,B 90.000,C 0.000} C_DIS
LIN {X 43.619,Y -42.046,Z -54.738,A -90.000,B 90.000,C 0.000} C_DIS
LIN {X 43.904,Y -42.037,Z -54.899,A -90.000,B 90.000,C 0.000} C_DIS
LIN {X 44.107,Y -42.033,Z -55.020,A -90.000,B 90.000,C 0.000} C_DIS
LIN {X 44.757,Y -42.006,Z -55.428,A -90.000,B 90.000,C 0.000} C_DIS
LIN {X 44.838,Y -42.001,Z -55.481,A -90.000,B 90.000,C 0.000} C_DIS
LIN {X 45.163,Y -41.988,Z -55.707,A -90.000,B 90.000,C 0.000} C_DIS
LIN {X 45.265,Y -41.985,Z -55.783,A -90.000,B 90.000,C 0.000} C_DIS
LIN {X 45.385,Y -41.991,Z -55.871,A -90.000,B 90.000,C 0.000} C_DIS
LIN {X 45.718,Y -42.018,Z -56.128,A -90.000,B 90.000,C 0.000} C_DIS
LIN {X 45.832,Y -42.025,Z -56.225,A -90.000,B 90.000,C 0.000} C_DIS
LIN {X 46.025,Y -42.047,Z -56.405,A -90.000,B 90.000,C 0.000} C_DIS
LIN {X 46.327,Y -42.112,Z -56.656,A -90.000,B 90.000,C 0.000} C_DIS
LIN {X 46.611,Y -42.224,Z -56.848,A -90.000,B 90.000,C 0.000} C_DIS
LIN {X 46.861,Y -42.332,Z -57.033,A -90.000,B 90.000,C 0.000} C_DIS
LIN {X 46.960,Y -42.379,Z -57.106,A -90.000,B 90.000,C 0.000} C_DIS
LIN {X 47.108,Y -42.456,Z -57.231,A -90.000,B 90.000,C 0.000} C_DIS
LIN {X 47.158,Y -42.479,Z -57.267,A -90.000,B 90.000,C 0.000} C_DIS
LIN {X 47.494,Y -42.476,Z -57.218,A -90.000,B 90.000,C 0.000} C_DIS
LIN {X 47.737,Y -42.475,Z -57.185,A -90.000,B 90.000,C 0.000} C_DIS
LIN {X 47.949,Y -42.480,Z -57.166,A -90.000,B 90.000,C 0.000} C_DIS
LIN {X 48.121,Y -42.482,Z -57.153,A -90.000,B 90.000,C 0.000} C_DIS
LIN {X 48.238,Y -42.484,Z -57.149,A -90.000,B 90.000,C 0.000} C_DIS
LIN {X 48.366,Y -42.487,Z -57.147,A -90.000,B 90.000,C 0.000} C_DIS
LIN {X 49.634,Y -42.480,Z -57.149,A -90.000,B 90.000,C 0.000} C_DIS
LIN {X 49.798,Y -42.480,Z -57.150,A -90.000,B 90.000,C 0.000} C_DIS
LIN {X 49.889,Y -42.482,Z -57.156,A -90.000,B 90.000,C 0.000} C_DIS
LIN {X 50.208,Y -42.482,Z -57.183,A -90.000,B 90.000,C 0.000} C_DIS
LIN {X 50.301,Y -42.478,Z -57.196,A -90.000,B 90.000,C 0.000} C_DIS
LIN {X 50.451,Y -42.476,Z -57.225,A -90.000,B 90.000,C 0.000} C_DIS
LIN {X 50.548,Y -42.476,Z -57.248,A -90.000,B 90.000,C 0.000} C_DIS
LIN {X 50.743,Y -42.466,Z -57.301,A -90.000,B 90.000,C 0.000} C_DIS
LIN {X 50.869,Y -42.460,Z -57.337,A -90.000,B 90.000,C 0.000} C_DIS
LIN {X 51.052,Y -42.458,Z -57.403,A -90.000,B 90.000,C 0.000} C_DIS
LIN {X 52.234,Y -42.482,Z -57.897,A -90.000,B 90.000,C 0.000} C_DIS
LIN {X 52.452,Y -42.482,Z -57.990,A -90.000,B 90.000,C 0.000} C_DIS
LIN {X 52.539,Y -42.478,Z -58.029,A -90.000,B 90.000,C 0.000} C_DIS
LIN {X 52.745,Y -42.463,Z -58.123,A -90.000,B 90.000,C 0.000} C_DIS
LIN {X 52.920,Y -42.440,Z -58.208,A -90.000,B 90.000,C 0.000} C_DIS
LIN {X 53.028,Y -42.426,Z -58.265,A -90.000,B 90.000,C 0.000} C_DIS
LIN {X 53.088,Y -42.417,Z -58.301,A -90.000,B 90.000,C 0.000} C_DIS
LIN {X 53.344,Y -42.385,Z -58.476,A -90.000,B 90.000,C 0.000} C_DIS
LIN {X 53.425,Y -42.372,Z -58.534,A -90.000,B 90.000,C 0.000} C_DIS
LIN {X 53.503,Y -42.360,Z -58.593,A -90.000,B 90.000,C 0.000} C_DIS
LIN {X 53.628,Y -42.348,Z -58.698,A -90.000,B 90.000,C 0.000} C_DIS
LIN {X 53.880,Y -42.330,Z -58.928,A -90.000,B 90.000,C 0.000} C_DIS
LIN {X 54.010,Y -42.324,Z -59.055,A -90.000,B 90.000,C 0.000} C_DIS
LIN {X 54.330,Y -42.314,Z -59.383,A -90.000,B 90.000,C 0.000} C_DIS
LIN {X 54.411,Y -42.313,Z -59.470,A -90.000,B 90.000,C 0.000} C_DIS
LIN {X 54.533,Y -42.315,Z -59.608,A -90.000,B 90.000,C 0.000} C_DIS
LIN {X 54.672,Y -42.317,Z -59.768,A -90.000,B 90.000,C 0.000} C_DIS
LIN {X 55.000,Y -42.330,Z -60.168,A -90.000,B 90.000,C 0.000} C_DIS
LIN {X 55.212,Y -42.325,Z -60.438,A -90.000,B 90.000,C 0.000} C_DIS
LIN {X 55.242,Y -42.322,Z -60.479,A -90.000,B 90.000,C 0.000} C_DIS
LIN {X 55.329,Y -42.318,Z -60.612,A -90.000,B 90.000,C 0.000} C_DIS
LIN {X 55.494,Y -42.317,Z -60.885,A -90.000,B 90.000,C 0.000} C_DIS
LIN {X 55.557,Y -42.319,Z -60.994,A -90.000,B 90.000,C 0.000} C_DIS
LIN {X 55.889,Y -42.342,Z -61.613,A -90.000,B 90.000,C 0.000} C_DIS
LIN {X 56.145,Y -42.357,Z -62.083,A -90.000,B 90.000,C 0.000} C_DIS
LIN {X 56.216,Y -42.363,Z -62.228,A -90.000,B 90.000,C 0.000} C_DIS
LIN {X 56.296,Y -42.373,Z -62.408,A -90.000,B 90.000,C 0.000} C_DIS
LIN {X 56.342,Y -42.371,Z -62.521,A -90.000,B 90.000,C 0.000} C_DIS
LIN {X 56.376,Y -42.371,Z -62.612,A -90.000,B 90.000,C 0.000} C_DIS
LIN {X 56.519,Y -42.377,Z -63.027,A -90.000,B 90.000,C 0.000} C_DIS
LIN {X 56.670,Y -42.378,Z -63.476,A -90.000,B 90.000,C 0.000} C_DIS
LIN {X 56.888,Y -42.373,Z -64.127,A -90.000,B 90.000,C 0.000} C_DIS
LIN {X 56.935,Y -42.372,Z -64.274,A -90.000,B 90.000,C 0.000} C_DIS
LIN {X 57.035,Y -42.379,Z -64.667,A -90.000,B 90.000,C 0.000} C_DIS
LIN {X 57.054,Y -42.382,Z -64.751,A -90.000,B 90.000,C 0.000} C_DIS
LIN {X 57.074,Y -42.388,Z -64.859,A -90.000,B 90.000,C 0.000} C_DIS
LIN {X 57.120,Y -42.422,Z -65.212,A -90.000,B 90.000,C 0.000} C_DIS
LIN {X 57.125,Y -42.425,Z -65.252,A -90.000,B 90.000,C 0.000} C_DIS
LIN {X 57.137,Y -42.440,Z -65.438,A -90.000,B 90.000,C 0.000} C_DIS
LIN {X 57.141,Y -42.454,Z -65.565,A -90.000,B 90.000,C 0.000} C_DIS
LIN {X 57.145,Y -42.473,Z -65.738,A -90.000,B 90.000,C 0.000} C_DIS
LIN {X 57.143,Y -42.486,Z -66.045,A -90.000,B 90.000,C 0.000} C_DIS
LIN {X 57.137,Y -42.489,Z -66.328,A -90.000,B 90.000,C 0.000} C_DIS
LIN {X 57.162,Y -42.479,Z -66.955,A -90.000,B 90.000,C 0.000} C_DIS
LIN {X 57.188,Y -42.489,Z -67.403,A -90.000,B 90.000,C 0.000} C_DIS
LIN {X 57.194,Y -42.497,Z -67.618,A -90.000,B 90.000,C 0.000} C_DIS
LIN {X 57.192,Y -42.507,Z -67.813,A -90.000,B 90.000,C 0.000} C_DIS
LIN {X 57.179,Y -42.520,Z -68.011,A -90.000,B 90.000,C 0.000} C_DIS
LIN {X 57.174,Y -42.523,Z -68.049,A -90.000,B 90.000,C 0.000} C_DIS
LIN {X 57.150,Y -42.528,Z -68.201,A -90.000,B 90.000,C 0.000} C_DIS
LIN {X 57.115,Y -42.534,Z -68.411,A -90.000,B 90.000,C 0.000} C_DIS
LIN {X 57.098,Y -42.533,Z -68.480,A -90.000,B 90.000,C 0.000} C_DIS
LIN {X 57.062,Y -42.535,Z -68.605,A -90.000,B 90.000,C 0.000} C_DIS
LIN {X 57.024,Y -42.538,Z -68.716,A -90.000,B 90.000,C 0.000} C_DIS
LIN {X 56.959,Y -42.537,Z -68.893,A -90.000,B 90.000,C 0.000} C_DIS
LIN {X 56.486,Y -42.607,Z -70.245,A -90.000,B 90.000,C 0.000} C_DIS
LIN {X 56.383,Y -42.609,Z -70.524,A -90.000,B 90.000,C 0.000} C_DIS
LIN {X 56.322,Y -42.601,Z -70.677,A -90.000,B 90.000,C 0.000} C_DIS
LIN {X 56.276,Y -42.595,Z -70.787,A -90.000,B 90.000,C 0.000} C_DIS
LIN {X 56.246,Y -42.588,Z -70.848,A -90.000,B 90.000,C 0.000} C_DIS
LIN {X 56.339,Y -42.631,Z -70.488,A -90.000,B 90.000,C 0.000} C_DIS
LIN {X 56.430,Y -42.642,Z -70.072,A -90.000,B 90.000,C 0.000} C_DIS
LIN {X 56.548,Y -42.640,Z -69.533,A -90.000,B 90.000,C 0.000} C_DIS
LIN {X 56.688,Y -42.649,Z -68.895,A -90.000,B 90.000,C 0.000} C_DIS
LIN {X 56.765,Y -42.669,Z -68.546,A -90.000,B 90.000,C 0.000} C_DIS
LIN {X 56.845,Y -42.666,Z -68.182,A -90.000,B 90.000,C 0.000} C_DIS
LIN {X 56.927,Y -42.629,Z -67.806,A -90.000,B 90.000,C 0.000} C_DIS
LIN {X 57.098,Y -42.513,Z -67.029,A -90.000,B 90.000,C 0.000} C_DIS
LIN {X 57.271,Y -42.425,Z -66.239,A -90.000,B 90.000,C 0.000} C_DIS
LIN {X 57.357,Y -42.376,Z -65.848,A -90.000,B 90.000,C 0.000} C_DIS
LIN {X 57.442,Y -42.291,Z -65.462,A -90.000,B 90.000,C 0.000} C_DIS
LIN {X 57.604,Y -42.079,Z -64.722,A -90.000,B 90.000,C 0.000} C_DIS
LIN {X 57.821,Y -41.805,Z -63.735,A -90.000,B 90.000,C 0.000} C_DIS
LIN {X 57.939,Y -41.644,Z -63.196,A -90.000,B 90.000,C 0.000} C_DIS
LIN {X 58.031,Y -41.471,Z -62.780,A -90.000,B 90.000,C 0.000} C_DIS
LIN {X 58.097,Y -41.308,Z -62.415,A -90.000,B 90.000,C 0.000} C_DIS
LIN {X 58.150,Y -41.319,Z -62.558,A -90.000,B 90.000,C 0.000} C_DIS
LIN {X 58.478,Y -41.378,Z -63.414,A -90.000,B 90.000,C 0.000} C_DIS
LIN {X 58.589,Y -41.383,Z -63.738,A -90.000,B 90.000,C 0.000} C_DIS
LIN {X 58.642,Y -41.385,Z -63.932,A -90.000,B 90.000,C 0.000} C_DIS
LIN {X 58.724,Y -41.390,Z -64.256,A -90.000,B 90.000,C 0.000} C_DIS
LIN {X 58.762,Y -41.397,Z -64.414,A -90.000,B 90.000,C 0.000} C_DIS
LIN {X 58.798,Y -41.408,Z -64.599,A -90.000,B 90.000,C 0.000} C_DIS
LIN {X 58.818,Y -41.419,Z -64.724,A -90.000,B 90.000,C 0.000} C_DIS
LIN {X 58.875,Y -41.461,Z -65.159,A -90.000,B 90.000,C 0.000} C_DIS
LIN {X 58.897,Y -41.490,Z -65.400,A -90.000,B 90.000,C 0.000} C_DIS
LIN {X 58.909,Y -41.519,Z -65.610,A -90.000,B 90.000,C 0.000} C_DIS
LIN {X 58.918,Y -41.550,Z -65.814,A -90.000,B 90.000,C 0.000} C_DIS
LIN {X 58.925,Y -41.570,Z -65.939,A -90.000,B 90.000,C 0.000} C_DIS
LIN {X 58.936,Y -41.607,Z -66.193,A -90.000,B 90.000,C 0.000} C_DIS
LIN {X 58.939,Y -41.619,Z -66.310,A -90.000,B 90.000,C 0.000} C_DIS
LIN {X 58.953,Y -41.632,Z -66.479,A -90.000,B 90.000,C 0.000} C_DIS
LIN {X 59.002,Y -41.650,Z -67.334,A -90.000,B 90.000,C 0.000} C_DIS
LIN {X 59.008,Y -41.656,Z -67.532,A -90.000,B 90.000,C 0.000} C_DIS
LIN {X 59.015,Y -41.673,Z -67.700,A -90.000,B 90.000,C 0.000} C_DIS
LIN {X 59.017,Y -41.702,Z -67.956,A -90.000,B 90.000,C 0.000} C_DIS
LIN {X 59.006,Y -41.738,Z -68.233,A -90.000,B 90.000,C 0.000} C_DIS
LIN {X 58.991,Y -41.761,Z -68.394,A -90.000,B 90.000,C 0.000} C_DIS
LIN {X 58.978,Y -41.771,Z -68.495,A -90.000,B 90.000,C 0.000} C_DIS
LIN {X 58.939,Y -41.796,Z -68.767,A -90.000,B 90.000,C 0.000} C_DIS
LIN {X 58.925,Y -41.805,Z -68.849,A -90.000,B 90.000,C 0.000} C_DIS
LIN {X 58.892,Y -41.814,Z -68.995,A -90.000,B 90.000,C 0.000} C_DIS
LIN {X 58.853,Y -41.820,Z -69.135,A -90.000,B 90.000,C 0.000} C_DIS
LIN {X 58.822,Y -41.825,Z -69.236,A -90.000,B 90.000,C 0.000} C_DIS
LIN {X 58.756,Y -41.834,Z -69.430,A -90.000,B 90.000,C 0.000} C_DIS
LIN {X 58.409,Y -41.963,Z -70.502,A -90.000,B 90.000,C 0.000} C_DIS
LIN {X 58.368,Y -41.974,Z -70.624,A -90.000,B 90.000,C 0.000} C_DIS
LIN {X 58.286,Y -41.987,Z -70.858,A -90.000,B 90.000,C 0.000} C_DIS
LIN {X 58.188,Y -41.988,Z -71.122,A -90.000,B 90.000,C 0.000} C_DIS
LIN {X 58.085,Y -41.974,Z -71.384,A -90.000,B 90.000,C 0.000} C_DIS
LIN {X 58.031,Y -41.963,Z -71.509,A -90.000,B 90.000,C 0.000} C_DIS
LIN {X 57.956,Y -41.962,Z -71.674,A -90.000,B 90.000,C 0.000} C_DIS
LIN {X 57.884,Y -41.963,Z -71.814,A -90.000,B 90.000,C 0.000} C_DIS
LIN {X 57.815,Y -41.965,Z -71.941,A -90.000,B 90.000,C 0.000} C_DIS
LIN {X 57.680,Y -41.970,Z -72.176,A -90.000,B 90.000,C 0.000} C_DIS
LIN {X 57.563,Y -41.976,Z -72.368,A -90.000,B 90.000,C 0.000} C_DIS
LIN {X 57.488,Y -41.981,Z -72.480,A -90.000,B 90.000,C 0.000} C_DIS
LIN {X 57.429,Y -41.986,Z -72.561,A -90.000,B 90.000,C 0.000} C_DIS
LIN {X 57.295,Y -41.996,Z -72.735,A -90.000,B 90.000,C 0.000} C_DIS
LIN {X 57.284,Y -41.996,Z -72.748,A -90.000,B 90.000,C 0.000} C_DIS
LIN {X 57.123,Y -41.995,Z -72.940,A -90.000,B 90.000,C 0.000} C_DIS
LIN {X 56.971,Y -41.993,Z -73.109,A -90.000,B 90.000,C 0.000} C_DIS
LIN {X 56.807,Y -41.985,Z -73.280,A -90.000,B 90.000,C 0.000} C_DIS
LIN {X 56.709,Y -41.971,Z -73.377,A -90.000,B 90.000,C 0.000} C_DIS
LIN {X 56.606,Y -41.959,Z -73.473,A -90.000,B 90.000,C 0.000} C_DIS
LIN {X 56.425,Y -41.940,Z -73.629,A -90.000,B 90.000,C 0.000} C_DIS
LIN {X 56.126,Y -41.903,Z -73.903,A -90.000,B 90.000,C 0.000} C_DIS
LIN {X 55.328,Y -41.834,Z -74.646,A -90.000,B 90.000,C 0.000} C_DIS
LIN {X 55.160,Y -41.818,Z -74.797,A -90.000,B 90.000,C 0.000} C_DIS
LIN {X 54.772,Y -41.759,Z -75.090,A -90.000,B 90.000,C 0.000} C_DIS
LIN {X 54.648,Y -41.743,Z -75.178,A -90.000,B 90.000,C 0.000} C_DIS
LIN {X 54.242,Y -41.693,Z -75.452,A -90.000,B 90.000,C 0.000} C_DIS
LIN {X 54.075,Y -41.677,Z -75.555,A -90.000,B 90.000,C 0.000} C_DIS
LIN {X 53.942,Y -41.666,Z -75.631,A -90.000,B 90.000,C 0.000} C_DIS
LIN {X 53.598,Y -41.641,Z -75.818,A -90.000,B 90.000,C 0.000} C_DIS
LIN {X 53.420,Y -41.632,Z -75.906,A -90.000,B 90.000,C 0.000} C_DIS
LIN {X 52.523,Y -41.597,Z -76.321,A -90.000,B 90.000,C 0.000} C_DIS
LIN {X 52.385,Y -41.594,Z -76.379,A -90.000,B 90.000,C 0.000} C_DIS
LIN {X 52.170,Y -41.592,Z -76.463,A -90.000,B 90.000,C 0.000} C_DIS
LIN {X 51.963,Y -41.587,Z -76.540,A -90.000,B 90.000,C 0.000} C_DIS
LIN {X 51.786,Y -41.585,Z -76.600,A -90.000,B 90.000,C 0.000} C_DIS
LIN {X 50.013,Y -41.584,Z -77.154,A -90.000,B 90.000,C 0.000} C_DIS
LIN {X 49.434,Y -41.572,Z -77.339,A -90.000,B 90.000,C 0.000} C_DIS
LIN {X 49.324,Y -41.571,Z -77.371,A -90.000,B 90.000,C 0.000} C_DIS
LIN {X 49.142,Y -41.574,Z -77.419,A -90.000,B 90.000,C 0.000} C_DIS
LIN {X 48.658,Y -41.588,Z -77.528,A -90.000,B 90.000,C 0.000} C_DIS
LIN {X 48.411,Y -41.599,Z -77.570,A -90.000,B 90.000,C 0.000} C_DIS
LIN {X 48.226,Y -41.608,Z -77.594,A -90.000,B 90.000,C 0.000} C_DIS
LIN {X 48.020,Y -41.616,Z -77.613,A -90.000,B 90.000,C 0.000} C_DIS
LIN {X 47.838,Y -41.624,Z -77.626,A -90.000,B 90.000,C 0.000} C_DIS
LIN {X 47.618,Y -41.640,Z -77.637,A -90.000,B 90.000,C 0.000} C_DIS
LIN {X 47.410,Y -41.659,Z -77.640,A -90.000,B 90.000,C 0.000} C_DIS
LIN {X 46.489,Y -41.751,Z -77.630,A -90.000,B 90.000,C 0.000} C_DIS
LIN {X 45.814,Y -41.788,Z -77.607,A -90.000,B 90.000,C 0.000} C_DIS
LIN {X 45.630,Y -41.797,Z -77.596,A -90.000,B 90.000,C 0.000} C_DIS
LIN {X 45.153,Y -41.816,Z -77.557,A -90.000,B 90.000,C 0.000} C_DIS
LIN {X 44.900,Y -41.842,Z -77.528,A -90.000,B 90.000,C 0.000} C_DIS
LIN {X 44.557,Y -41.881,Z -77.476,A -90.000,B 90.000,C 0.000} C_DIS
LIN {X 44.490,Y -41.890,Z -77.465,A -90.000,B 90.000,C 0.000} C_DIS
LIN {X 44.265,Y -41.904,Z -77.412,A -90.000,B 90.000,C 0.000} C_DIS
LIN {X 43.864,Y -41.935,Z -77.297,A -90.000,B 90.000,C 0.000} C_DIS
LIN {X 43.449,Y -41.958,Z -77.173,A -90.000,B 90.000,C 0.000} C_DIS
LIN {X 43.233,Y -41.966,Z -77.106,A -90.000,B 90.000,C 0.000} C_DIS
LIN {X 43.060,Y -41.969,Z -77.053,A -90.000,B 90.000,C 0.000} C_DIS
LIN {X 42.852,Y -41.973,Z -76.991,A -90.000,B 90.000,C 0.000} C_DIS
LIN {X 42.648,Y -41.978,Z -76.924,A -90.000,B 90.000,C 0.000} C_DIS
LIN {X 42.476,Y -41.985,Z -76.860,A -90.000,B 90.000,C 0.000} C_DIS
LIN {X 42.178,Y -41.986,Z -76.739,A -90.000,B 90.000,C 0.000} C_DIS
LIN {X 41.751,Y -41.914,Z -76.873,A -90.000,B 90.000,C 0.000} C_DIS
LIN {X 41.504,Y -41.870,Z -76.945,A -90.000,B 90.000,C 0.000} C_DIS
LIN {X 41.325,Y -41.837,Z -76.993,A -90.000,B 90.000,C 0.000} C_DIS
LIN {X 40.985,Y -41.809,Z -77.094,A -90.000,B 90.000,C 0.000} C_DIS
LIN {X 40.702,Y -41.784,Z -77.170,A -90.000,B 90.000,C 0.000} C_DIS
LIN {X 40.591,Y -41.775,Z -77.196,A -90.000,B 90.000,C 0.000} C_DIS
LIN {X 40.456,Y -41.763,Z -77.226,A -90.000,B 90.000,C 0.000} C_DIS
LIN {X 40.015,Y -41.720,Z -77.344,A -90.000,B 90.000,C 0.000} C_DIS
LIN {X 39.633,Y -41.677,Z -77.427,A -90.000,B 90.000,C 0.000} C_DIS
LIN {X 39.251,Y -41.661,Z -77.501,A -90.000,B 90.000,C 0.000} C_DIS
LIN {X 38.769,Y -41.628,Z -77.586,A -90.000,B 90.000,C 0.000} C_DIS
LIN {X 38.474,Y -41.607,Z -77.634,A -90.000,B 90.000,C 0.000} C_DIS
LIN {X 38.367,Y -41.599,Z -77.647,A -90.000,B 90.000,C 0.000} C_DIS
LIN {X 38.181,Y -41.584,Z -77.664,A -90.000,B 90.000,C 0.000} C_DIS
LIN {X 38.018,Y -41.569,Z -77.672,A -90.000,B 90.000,C 0.000} C_DIS
LIN {X 37.924,Y -41.560,Z -77.675,A -90.000,B 90.000,C 0.000} C_DIS
LIN {X 37.603,Y -41.513,Z -77.678,A -90.000,B 90.000,C 0.000} C_DIS
LIN {X 37.324,Y -41.470,Z -77.674,A -90.000,B 90.000,C 0.000} C_DIS
LIN {X 37.270,Y -41.462,Z -77.673,A -90.000,B 90.000,C 0.000} C_DIS
LIN {X 36.864,Y -41.421,Z -77.678,A -90.000,B 90.000,C 0.000} C_DIS
LIN {X 36.743,Y -41.402,Z -77.676,A -90.000,B 90.000,C 0.000} C_DIS
LIN {X 36.551,Y -41.370,Z -77.666,A -90.000,B 90.000,C 0.000} C_DIS
LIN {X 36.410,Y -41.343,Z -77.651,A -90.000,B 90.000,C 0.000} C_DIS
LIN {X 36.245,Y -41.308,Z -77.624,A -90.000,B 90.000,C 0.000} C_DIS
LIN {X 36.068,Y -41.275,Z -77.594,A -90.000,B 90.000,C 0.000} C_DIS
LIN {X 35.898,Y -41.238,Z -77.562,A -90.000,B 90.000,C 0.000} C_DIS
LIN {X 35.736,Y -41.230,Z -77.528,A -90.000,B 90.000,C 0.000} C_DIS
LIN {X 35.294,Y -41.262,Z -77.424,A -90.000,B 90.000,C 0.000} C_DIS
LIN {X 35.037,Y -41.284,Z -77.359,A -90.000,B 90.000,C 0.000} C_DIS
LIN {X 34.811,Y -41.299,Z -77.300,A -90.000,B 90.000,C 0.000} C_DIS
LIN {X 34.615,Y -41.301,Z -77.252,A -90.000,B 90.000,C 0.000} C_DIS
LIN {X 34.529,Y -41.300,Z -77.234,A -90.000,B 90.000,C 0.000} C_DIS
LIN {X 34.414,Y -41.296,Z -77.215,A -90.000,B 90.000,C 0.000} C_DIS
LIN {X 34.316,Y -41.287,Z -77.208,A -90.000,B 90.000,C 0.000} C_DIS
LIN {X 34.260,Y -41.279,Z -77.211,A -90.000,B 90.000,C 0.000} C_DIS
LIN {X 34.213,Y -41.268,Z -77.220,A -90.000,B 90.000,C 0.000} C_DIS
LIN {X 34.173,Y -41.254,Z -77.236,A -90.000,B 90.000,C 0.000} C_DIS
LIN {X 34.140,Y -41.239,Z -77.259,A -90.000,B 90.000,C 0.000} C_DIS
LIN {X 34.116,Y -41.222,Z -77.290,A -90.000,B 90.000,C 0.000} C_DIS
LIN {X 34.099,Y -41.204,Z -77.330,A -90.000,B 90.000,C 0.000} C_DIS
LIN {X 34.091,Y -41.183,Z -77.379,A -90.000,B 90.000,C 0.000} C_DIS
LIN {X 34.090,Y -41.159,Z -77.438,A -90.000,B 90.000,C 0.000} C_DIS
LIN {X 34.103,Y -41.115,Z -77.544,A -90.000,B 90.000,C 0.000} C_DIS
LIN {X 34.134,Y -41.062,Z -77.675,A -90.000,B 90.000,C 0.000} C_DIS
LIN {X 34.149,Y -41.052,Z -77.725,A -90.000,B 90.000,C 0.000} C_DIS
LIN {X 34.203,Y -41.124,Z -77.891,A -90.000,B 90.000,C 0.000} C_DIS
LIN {X 34.250,Y -41.179,Z -78.018,A -90.000,B 90.000,C 0.000} C_DIS
LIN {X 34.367,Y -41.308,Z -78.311,A -90.000,B 90.000,C 0.000} C_DIS
LIN {X 34.422,Y -41.368,Z -78.444,A -90.000,B 90.000,C 0.000} C_DIS
LIN {X 34.479,Y -41.418,Z -78.555,A -90.000,B 90.000,C 0.000} C_DIS
LIN {X 34.507,Y -41.441,Z -78.605,A -90.000,B 90.000,C 0.000} C_DIS
LIN {X 34.554,Y -41.469,Z -78.680,A -90.000,B 90.000,C 0.000} C_DIS
LIN {X 34.596,Y -41.492,Z -78.741,A -90.000,B 90.000,C 0.000} C_DIS
LIN {X 34.664,Y -41.526,Z -78.829,A -90.000,B 90.000,C 0.000} C_DIS
LIN {X 34.761,Y -41.569,Z -78.940,A -90.000,B 90.000,C 0.000} C_DIS
LIN {X 34.877,Y -41.615,Z -79.050,A -90.000,B 90.000,C 0.000} C_DIS
LIN {X 35.013,Y -41.669,Z -79.158,A -90.000,B 90.000,C 0.000} C_DIS
LIN {X 35.110,Y -41.696,Z -79.224,A -90.000,B 90.000,C 0.000} C_DIS
LIN {X 35.235,Y -41.728,Z -79.299,A -90.000,B 90.000,C 0.000} C_DIS
LIN {X 35.269,Y -41.736,Z -79.317,A -90.000,B 90.000,C 0.000} C_DIS
LIN {X 35.460,Y -41.776,Z -79.403,A -90.000,B 90.000,C 0.000} C_DIS
LIN {X 35.619,Y -41.805,Z -79.458,A -90.000,B 90.000,C 0.000} C_DIS
LIN {X 35.758,Y -41.818,Z -79.496,A -90.000,B 90.000,C 0.000} C_DIS
LIN {X 35.997,Y -41.837,Z -79.545,A -90.000,B 90.000,C 0.000} C_DIS
LIN {X 36.108,Y -41.845,Z -79.564,A -90.000,B 90.000,C 0.000} C_DIS
LIN {X 36.253,Y -41.855,Z -79.584,A -90.000,B 90.000,C 0.000} C_DIS
LIN {X 36.387,Y -41.863,Z -79.598,A -90.000,B 90.000,C 0.000} C_DIS
LIN {X 36.570,Y -41.873,Z -79.612,A -90.000,B 90.000,C 0.000} C_DIS
LIN {X 36.765,Y -41.875,Z -79.623,A -90.000,B 90.000,C 0.000} C_DIS
LIN {X 37.182,Y -41.877,Z -79.629,A -90.000,B 90.000,C 0.000} C_DIS
LIN {X 37.521,Y -41.879,Z -79.643,A -90.000,B 90.000,C 0.000} C_DIS
LIN {X 37.901,Y -41.882,Z -79.649,A -90.000,B 90.000,C 0.000} C_DIS
LIN {X 37.992,Y -41.883,Z -79.648,A -90.000,B 90.000,C 0.000} C_DIS
LIN {X 38.173,Y -41.885,Z -79.643,A -90.000,B 90.000,C 0.000} C_DIS
LIN {X 38.408,Y -41.885,Z -79.628,A -90.000,B 90.000,C 0.000} C_DIS
LIN {X 38.583,Y -41.885,Z -79.614,A -90.000,B 90.000,C 0.000} C_DIS
LIN {X 38.773,Y -41.884,Z -79.592,A -90.000,B 90.000,C 0.000} C_DIS
LIN {X 39.087,Y -41.880,Z -79.544,A -90.000,B 90.000,C 0.000} C_DIS
LIN {X 39.627,Y -41.866,Z -79.454,A -90.000,B 90.000,C 0.000} C_DIS
LIN {X 40.002,Y -41.858,Z -79.385,A -90.000,B 90.000,C 0.000} C_DIS
LIN {X 40.425,Y -41.849,Z -79.297,A -90.000,B 90.000,C 0.000} C_DIS
LIN {X 40.498,Y -41.847,Z -79.281,A -90.000,B 90.000,C 0.000} C_DIS
LIN {X 40.926,Y -41.836,Z -79.169,A -90.000,B 90.000,C 0.000} C_DIS
LIN {X 41.157,Y -41.829,Z -79.117,A -90.000,B 90.000,C 0.000} C_DIS
LIN {X 41.566,Y -41.814,Z -79.008,A -90.000,B 90.000,C 0.000} C_DIS
LIN {X 41.908,Y -41.798,Z -78.906,A -90.000,B 90.000,C 0.000} C_DIS
LIN {X 42.011,Y -41.793,Z -78.878,A -90.000,B 90.000,C 0.000} C_DIS
LIN {X 42.120,Y -41.788,Z -78.846,A -90.000,B 90.000,C 0.000} C_DIS
LIN {X 42.196,Y -41.783,Z -78.871,A -90.000,B 90.000,C 0.000} C_DIS
LIN {X 42.392,Y -41.768,Z -78.930,A -90.000,B 90.000,C 0.000} C_DIS
LIN {X 42.665,Y -41.747,Z -79.012,A -90.000,B 90.000,C 0.000} C_DIS
LIN {X 43.282,Y -41.700,Z -79.196,A -90.000,B 90.000,C 0.000} C_DIS
LIN {X 43.533,Y -41.681,Z -79.268,A -90.000,B 90.000,C 0.000} C_DIS
LIN {X 43.614,Y -41.678,Z -79.292,A -90.000,B 90.000,C 0.000} C_DIS
LIN {X 43.738,Y -41.671,Z -79.327,A -90.000,B 90.000,C 0.000} C_DIS
LIN {X 44.023,Y -41.646,Z -79.394,A -90.000,B 90.000,C 0.000} C_DIS
LIN {X 44.156,Y -41.635,Z -79.420,A -90.000,B 90.000,C 0.000} C_DIS
LIN {X 44.593,Y -41.601,Z -79.490,A -90.000,B 90.000,C 0.000} C_DIS
LIN {X 44.803,Y -41.575,Z -79.514,A -90.000,B 90.000,C 0.000} C_DIS
LIN {X 44.902,Y -41.566,Z -79.526,A -90.000,B 90.000,C 0.000} C_DIS
LIN {X 45.457,Y -41.515,Z -79.569,A -90.000,B 90.000,C 0.000} C_DIS
LIN {X 45.632,Y -41.500,Z -79.574,A -90.000,B 90.000,C 0.000} C_DIS
LIN {X 45.731,Y -41.491,Z -79.583,A -90.000,B 90.000,C 0.000} C_DIS
LIN {X 46.365,Y -41.434,Z -79.601,A -90.000,B 90.000,C 0.000} C_DIS
LIN {X 47.145,Y -41.365,Z -79.612,A -90.000,B 90.000,C 0.000} C_DIS
LIN {X 47.362,Y -41.343,Z -79.614,A -90.000,B 90.000,C 0.000} C_DIS
LIN {X 47.653,Y -41.308,Z -79.609,A -90.000,B 90.000,C 0.000} C_DIS
LIN {X 47.653,Y -60.000,Z -79.609,A -90.000,B 90.000,C 0.000} C_DIS
LIN {X 60.545,Y -60.000,Z -70.157,A -90.000,B 90.000,C 0.000} C_DIS
LIN {X 60.545,Y -41.308,Z -70.157,A -90.000,B 90.000,C 0.000} C_DIS
LIN {X 60.360,Y -41.438,Z -70.776,A -90.000,B 90.000,C 0.000} C_DIS
LIN {X 60.290,Y -41.481,Z -71.006,A -90.000,B 90.000,C 0.000} C_DIS
LIN {X 60.239,Y -41.509,Z -71.170,A -90.000,B 90.000,C 0.000} C_DIS
LIN {X 60.174,Y -41.529,Z -71.363,A -90.000,B 90.000,C 0.000} C_DIS
LIN {X 60.107,Y -41.540,Z -71.555,A -90.000,B 90.000,C 0.000} C_DIS
LIN {X 60.026,Y -41.543,Z -71.775,A -90.000,B 90.000,C 0.000} C_DIS
LIN {X 59.966,Y -41.539,Z -71.930,A -90.000,B 90.000,C 0.000} C_DIS
LIN {X 59.869,Y -41.553,Z -72.186,A -90.000,B 90.000,C 0.000} C_DIS
LIN {X 59.816,Y -41.561,Z -72.316,A -90.000,B 90.000,C 0.000} C_DIS
LIN {X 59.743,Y -41.572,Z -72.483,A -90.000,B 90.000,C 0.000} C_DIS
LIN {X 59.697,Y -41.579,Z -72.580,A -90.000,B 90.000,C 0.000} C_DIS
LIN {X 59.554,Y -41.600,Z -72.859,A -90.000,B 90.000,C 0.000} C_DIS
LIN {X 59.402,Y -41.623,Z -73.133,A -90.000,B 90.000,C 0.000} C_DIS
LIN {X 59.318,Y -41.629,Z -73.275,A -90.000,B 90.000,C 0.000} C_DIS
LIN {X 59.221,Y -41.628,Z -73.431,A -90.000,B 90.000,C 0.000} C_DIS
LIN {X 59.080,Y -41.620,Z -73.636,A -90.000,B 90.000,C 0.000} C_DIS
LIN {X 59.058,Y -41.618,Z -73.664,A -90.000,B 90.000,C 0.000} C_DIS
LIN {X 58.951,Y -41.609,Z -73.804,A -90.000,B 90.000,C 0.000} C_DIS
LIN {X 58.824,Y -41.591,Z -73.958,A -90.000,B 90.000,C 0.000} C_DIS
LIN {X 58.577,Y -41.559,Z -74.242,A -90.000,B 90.000,C 0.000} C_DIS
LIN {X 58.361,Y -41.535,Z -74.472,A -90.000,B 90.000,C 0.000} C_DIS
LIN {X 58.066,Y -41.504,Z -74.770,A -90.000,B 90.000,C 0.000} C_DIS
LIN {X 57.960,Y -41.494,Z -74.870,A -90.000,B 90.000,C 0.000} C_DIS
LIN {X 57.886,Y -41.486,Z -74.935,A -90.000,B 90.000,C 0.000} C_DIS
LIN {X 57.761,Y -41.472,Z -75.041,A -90.000,B 90.000,C 0.000} C_DIS
LIN {X 57.531,Y -41.443,Z -75.253,A -90.000,B 90.000,C 0.000} C_DIS
LIN {X 57.277,Y -41.398,Z -75.481,A -90.000,B 90.000,C 0.000} C_DIS
LIN {X 56.794,Y -41.308,Z -75.913,A -90.000,B 90.000,C 0.000} C_DIS
LIN {X 56.610,Y -41.279,Z -76.076,A -90.000,B 90.000,C 0.000} C_DIS
LIN {X 56.447,Y -41.248,Z -76.218,A -90.000,B 90.000,C 0.000} C_DIS
LIN {X 56.306,Y -41.223,Z -76.338,A -90.000,B 90.000,C 0.000} C_DIS
LIN {X 56.085,Y -41.185,Z -76.518,A -90.000,B 90.000,C 0.000} C_DIS
LIN {X 56.003,Y -41.172,Z -76.580,A -90.000,B 90.000,C 0.000} C_DIS
LIN {X 55.916,Y -41.161,Z -76.638,A -90.000,B 90.000,C 0.000} C_DIS
LIN {X 55.879,Y -41.158,Z -76.655,A -90.000,B 90.000,C 0.000} C_DIS
LIN {X 55.868,Y -41.158,Z -76.657,A -90.000,B 90.000,C 0.000} C_DIS
LIN {X 55.858,Y -41.159,Z -76.653,A -90.000,B 90.000,C 0.000} C_DIS
LIN {X 55.857,Y -41.163,Z -76.641,A -90.000,B 90.000,C 0.000} C_DIS
LIN {X 55.869,Y -41.170,Z -76.611,A -90.000,B 90.000,C 0.000} C_DIS
LIN {X 55.916,Y -41.188,Z -76.540,A -90.000,B 90.000,C 0.000} C_DIS
LIN {X 56.027,Y -41.220,Z -76.401,A -90.000,B 90.000,C 0.000} C_DIS
LIN {X 56.188,Y -41.263,Z -76.215,A -90.000,B 90.000,C 0.000} C_DIS
LIN {X 56.513,Y -41.343,Z -75.863,A -90.000,B 90.000,C 0.000} C_DIS
LIN {X 56.778,Y -41.403,Z -75.587,A -90.000,B 90.000,C 0.000} C_DIS
LIN {X 57.074,Y -41.467,Z -75.287,A -90.000,B 90.000,C 0.000} C_DIS
LIN {X 57.233,Y -41.495,Z -75.129,A -90.000,B 90.000,C 0.000} C_DIS
LIN {X 57.398,Y -41.518,Z -74.966,A -90.000,B 90.000,C 0.000} C_DIS
LIN {X 57.743,Y -41.564,Z -74.632,A -90.000,B 90.000,C 0.000} C_DIS
LIN {X 57.923,Y -41.585,Z -74.462,A -90.000,B 90.000,C 0.000} C_DIS
LIN {X 58.478,Y -41.631,Z -73.948,A -90.000,B 90.000,C 0.000} C_DIS
LIN {X 58.667,Y -41.646,Z -73.777,A -90.000,B 90.000,C 0.000} C_DIS
LIN {X 58.857,Y -41.656,Z -73.608,A -90.000,B 90.000,C 0.000} C_DIS
LIN {X 59.047,Y -41.656,Z -73.442,A -90.000,B 90.000,C 0.000} C_DIS
LIN {X 59.236,Y -41.645,Z -73.279,A -90.000,B 90.000,C 0.000} C_DIS
LIN {X 59.424,Y -41.623,Z -73.121,A -90.000,B 90.000,C 0.000} C_DIS
LIN {X 59.611,Y -41.597,Z -72.966,A -90.000,B 90.000,C 0.000} C_DIS
LIN {X 59.795,Y -41.565,Z -72.818,A -90.000,B 90.000,C 0.000} C_DIS
LIN {X 60.152,Y -41.508,Z -72.540,A -90.000,B 90.000,C 0.000} C_DIS
LIN {X 60.492,Y -41.455,Z -72.293,A -90.000,B 90.000,C 0.000} C_DIS
LIN {X 60.732,Y -41.417,Z -72.131,A -90.000,B 90.000,C 0.000} C_DIS
LIN {X 60.884,Y -41.393,Z -72.036,A -90.000,B 90.000,C 0.000} C_DIS
LIN {X 61.028,Y -41.371,Z -71.953,A -90.000,B 90.000,C 0.000} C_DIS
LIN {X 61.229,Y -41.336,Z -71.849,A -90.000,B 90.000,C 0.000} C_DIS
LIN {X 61.352,Y -41.313,Z -71.796,A -90.000,B 90.000,C 0.000} C_DIS
LIN {X 61.465,Y -41.290,Z -71.757,A -90.000,B 90.000,C 0.000} C_DIS
LIN {X 61.568,Y -41.268,Z -71.732,A -90.000,B 90.000,C 0.000} C_DIS
LIN {X 61.615,Y -41.258,Z -71.725,A -90.000,B 90.000,C 0.000} C_DIS
LIN {X 61.681,Y -41.245,Z -71.722,A -90.000,B 90.000,C 0.000} C_DIS
LIN {X 61.721,Y -41.237,Z -71.725,A -90.000,B 90.000,C 0.000} C_DIS
LIN {X 61.758,Y -41.230,Z -71.732,A -90.000,B 90.000,C 0.000} C_DIS
LIN {X 61.792,Y -41.224,Z -71.743,A -90.000,B 90.000,C 0.000} C_DIS
LIN {X 61.822,Y -41.219,Z -71.758,A -90.000,B 90.000,C 0.000} C_DIS
LIN {X 61.850,Y -41.215,Z -71.778,A -90.000,B 90.000,C 0.000} C_DIS
LIN {X 61.873,Y -41.213,Z -71.803,A -90.000,B 90.000,C 0.000} C_DIS
LIN {X 61.894,Y -41.211,Z -71.832,A -90.000,B 90.000,C 0.000} C_DIS
LIN {X 61.911,Y -41.210,Z -71.865,A -90.000,B 90.000,C 0.000} C_DIS
LIN {X 61.929,Y -41.211,Z -71.925,A -90.000,B 90.000,C 0.000} C_DIS
LIN {X 61.937,Y -41.213,Z -71.970,A -90.000,B 90.000,C 0.000} C_DIS
LIN {X 61.941,Y -41.215,Z -72.021,A -90.000,B 90.000,C 0.000} C_DIS
LIN {X 61.941,Y -41.218,Z -72.077,A -90.000,B 90.000,C 0.000} C_DIS
LIN {X 61.929,Y -41.224,Z -72.204,A -90.000,B 90.000,C 0.000} C_DIS
LIN {X 61.900,Y -41.230,Z -72.352,A -90.000,B 90.000,C 0.000} C_DIS
LIN {X 61.854,Y -41.236,Z -72.523,A -90.000,B 90.000,C 0.000} C_DIS
LIN {X 61.824,Y -41.249,Z -72.617,A -90.000,B 90.000,C 0.000} C_DIS
LIN {X 61.751,Y -41.277,Z -72.822,A -90.000,B 90.000,C 0.000} C_DIS
LIN {X 61.659,Y -41.308,Z -73.051,A -90.000,B 90.000,C 0.000} C_DIS
LIN {X 61.547,Y -41.348,Z -73.317,A -90.000,B 90.000,C 0.000} C_DIS
LIN {X 61.461,Y -41.377,Z -73.502,A -90.000,B 90.000,C 0.000} C_DIS
LIN {X 61.393,Y -41.398,Z -73.635,A -90.000,B 90.000,C 0.000} C_DIS
LIN {X 61.334,Y -41.412,Z -73.752,A -90.000,B 90.000,C 0.000} C_DIS
LIN {X 61.265,Y -41.421,Z -73.880,A -90.000,B 90.000,C 0.000} C_DIS
LIN {X 61.141,Y -41.428,Z -74.101,A -90.000,B 90.000,C 0.000} C_DIS
LIN {X 61.030,Y -41.426,Z -74.289,A -90.000,B 90.000,C 0.000} C_DIS
LIN {X 60.948,Y -41.420,Z -74.420,A -90.000,B 90.000,C 0.000} C_DIS
LIN {X 60.890,Y -41.413,Z -74.511,A -90.000,B 90.000,C 0.000} C_DIS
LIN {X 60.697,Y -41.382,Z -74.787,A -90.000,B 90.000,C 0.000} C_DIS
LIN {X 60.609,Y -41.369,Z -74.903,A -90.000,B 90.000,C 0.000} C_DIS
LIN {X 60.498,Y -41.353,Z -75.045,A -90.000,B 90.000,C 0.000} C_DIS
LIN {X 60.334,Y -41.332,Z -75.244,A -90.000,B 90.000,C 0.000} C_DIS
LIN {X 60.144,Y -41.308,Z -75.462,A -90.000,B 90.000,C 0.000} C_DIS
LIN {X 59.976,Y -41.286,Z -75.660,A -90.000,B 90.000,C 0.000} C_DIS
LIN {X 59.910,Y -41.275,Z -75.741,A -90.000,B 90.000,C 0.000} C_DIS
LIN {X 59.811,Y -41.255,Z -75.870,A -90.000,B 90.000,C 0.000} C_DIS
LIN {X 59.778,Y -41.248,Z -75.919,A -90.000,B 90.000,C 0.000} C_DIS
LIN {X 59.748,Y -41.240,Z -75.974,A -90.000,B 90.000,C 0.000} C_DIS
LIN {X 59.739,Y -41.236,Z -75.999,A -90.000,B 90.000,C 0.000} C_DIS
LIN {X 59.739,Y -41.235,Z -76.009,A -90.000,B 90.000,C 0.000} C_DIS
LIN {X 59.745,Y -41.233,Z -76.020,A -90.000,B 90.000,C 0.000} C_DIS
LIN {X 59.759,Y -41.232,Z -76.024,A -90.000,B 90.000,C 0.000} C_DIS
LIN {X 59.782,Y -41.232,Z -76.019,A -90.000,B 90.000,C 0.000} C_DIS
LIN {X 59.851,Y -41.236,Z -75.987,A -90.000,B 90.000,C 0.000} C_DIS
LIN {X 59.950,Y -41.243,Z -75.929,A -90.000,B 90.000,C 0.000} C_DIS
LIN {X 60.074,Y -41.254,Z -75.846,A -90.000,B 90.000,C 0.000} C_DIS
LIN {X 60.221,Y -41.266,Z -75.742,A -90.000,B 90.000,C 0.000} C_DIS
LIN {X 60.572,Y -41.288,Z -75.485,A -90.000,B 90.000,C 0.000} C_DIS
LIN {X 60.979,Y -41.323,Z -75.183,A -90.000,B 90.000,C 0.000} C_DIS
LIN {X 61.196,Y -41.347,Z -75.023,A -90.000,B 90.000,C 0.000} C_DIS
LIN {X 61.417,Y -41.364,Z -74.860,A -90.000,B 90.000,C 0.000} C_DIS
LIN {X 61.641,Y -41.378,Z -74.699,A -90.000,B 90.000,C 0.000} C_DIS
LIN {X 61.863,Y -41.383,Z -74.543,A -90.000,B 90.000,C 0.000} C_DIS
LIN {X 62.081,Y -41.375,Z -74.393,A -90.000,B 90.000,C 0.000} C_DIS
LIN {X 62.187,Y -41.367,Z -74.323,A -90.000,B 90.000,C 0.000} C_DIS
LIN {X 62.393,Y -41.345,Z -74.191,A -90.000,B 90.000,C 0.000} C_DIS
LIN {X 62.588,Y -41.316,Z -74.074,A -90.000,B 90.000,C 0.000} C_DIS
LIN {X 62.679,Y -41.299,Z -74.023,A -90.000,B 90.000,C 0.000} C_DIS
LIN {X 62.850,Y -41.266,Z -73.935,A -90.000,B 90.000,C 0.000} C_DIS
LIN {X 62.929,Y -41.250,Z -73.900,A -90.000,B 90.000,C 0.000} C_DIS
LIN {X 63.036,Y -41.227,Z -73.859,A -90.000,B 90.000,C 0.000} C_DIS
LIN {X 63.101,Y -41.214,Z -73.840,A -90.000,B 90.000,C 0.000} C_DIS
LIN {X 63.159,Y -41.204,Z -73.829,A -90.000,B 90.000,C 0.000} C_DIS
LIN {X 63.211,Y -41.196,Z -73.824,A -90.000,B 90.000,C 0.000} C_DIS
LIN {X 63.257,Y -41.201,Z -73.828,A -90.000,B 90.000,C 0.000} C_DIS
LIN {X 63.294,Y -41.208,Z -73.841,A -90.000,B 90.000,C 0.000} C_DIS
LIN {X 63.325,Y -41.216,Z -73.862,A -90.000,B 90.000,C 0.000} C_DIS
LIN {X 63.347,Y -41.224,Z -73.892,A -90.000,B 90.000,C 0.000} C_DIS
LIN {X 63.360,Y -41.233,Z -73.932,A -90.000,B 90.000,C 0.000} C_DIS
LIN {X 63.365,Y -41.242,Z -73.981,A -90.000,B 90.000,C 0.000} C_DIS
LIN {X 63.361,Y -41.251,Z -74.042,A -90.000,B 90.000,C 0.000} C_DIS
LIN {X 63.347,Y -41.261,Z -74.112,A -90.000,B 90.000,C 0.000} C_DIS
LIN {X 63.323,Y -41.271,Z -74.194,A -90.000,B 90.000,C 0.000} C_DIS
LIN {X 63.268,Y -41.286,Z -74.339,A -90.000,B 90.000,C 0.000} C_DIS
LIN {X 63.218,Y -41.297,Z -74.451,A -90.000,B 90.000,C 0.000} C_DIS
LIN {X 63.157,Y -41.308,Z -74.575,A -90.000,B 90.000,C 0.000} C_DIS
LIN {X 63.091,Y -41.320,Z -74.703,A -90.000,B 90.000,C 0.000} C_DIS
LIN {X 62.957,Y -41.340,Z -74.947,A -90.000,B 90.000,C 0.000} C_DIS
LIN {X 62.875,Y -41.341,Z -75.093,A -90.000,B 90.000,C 0.000} C_DIS
LIN {X 62.821,Y -41.337,Z -75.185,A -90.000,B 90.000,C 0.000} C_DIS
LIN {X 62.687,Y -41.319,Z -75.406,A -90.000,B 90.000,C 0.000} C_DIS
LIN {X 62.610,Y -41.308,Z -75.528,A -90.000,B 90.000,C 0.000} C_DIS
LIN {X 62.564,Y -41.307,Z -75.607,A -90.000,B 90.000,C 0.000} C_DIS
LIN {X 62.519,Y -41.301,Z -75.685,A -90.000,B 90.000,C 0.000} C_DIS
LIN {X 62.438,Y -41.288,Z -75.838,A -90.000,B 90.000,C 0.000} C_DIS
LIN {X 62.370,Y -41.275,Z -75.987,A -90.000,B 90.000,C 0.000} C_DIS
LIN {X 62.312,Y -41.264,Z -76.132,A -90.000,B 90.000,C 0.000} C_DIS
LIN {X 62.267,Y -41.256,Z -76.272,A -90.000,B 90.000,C 0.000} C_DIS
LIN {X 62.233,Y -41.249,Z -76.407,A -90.000,B 90.000,C 0.000} C_DIS
LIN {X 62.209,Y -41.242,Z -76.537,A -90.000,B 90.000,C 0.000} C_DIS
LIN {X 62.202,Y -41.240,Z -76.600,A -90.000,B 90.000,C 0.000} C_DIS
LIN {X 62.194,Y -41.235,Z -76.721,A -90.000,B 90.000,C 0.000} C_DIS
LIN {X 62.196,Y -41.231,Z -76.836,A -90.000,B 90.000,C 0.000} C_DIS
LIN {X 62.208,Y -41.228,Z -76.944,A -90.000,B 90.000,C 0.000} C_DIS
LIN {X 62.228,Y -41.226,Z -77.044,A -90.000,B 90.000,C 0.000} C_DIS
LIN {X 62.242,Y -41.225,Z -77.092,A -90.000,B 90.000,C 0.000} C_DIS
LIN {X 62.275,Y -41.224,Z -77.181,A -90.000,B 90.000,C 0.000} C_DIS
LIN {X 62.317,Y -41.224,Z -77.263,A -90.000,B 90.000,C 0.000} C_DIS
LIN {X 62.341,Y -41.224,Z -77.300,A -90.000,B 90.000,C 0.000} C_DIS
LIN {X 62.394,Y -41.225,Z -77.369,A -90.000,B 90.000,C 0.000} C_DIS
LIN {X 62.455,Y -41.226,Z -77.428,A -90.000,B 90.000,C 0.000} C_DIS
LIN {X 62.488,Y -41.227,Z -77.454,A -90.000,B 90.000,C 0.000} C_DIS
LIN {X 62.559,Y -41.230,Z -77.499,A -90.000,B 90.000,C 0.000} C_DIS
LIN {X 62.636,Y -41.233,Z -77.534,A -90.000,B 90.000,C 0.000} C_DIS
LIN {X 62.720,Y -41.236,Z -77.559,A -90.000,B 90.000,C 0.000} C_DIS
LIN {X 62.809,Y -41.240,Z -77.573,A -90.000,B 90.000,C 0.000} C_DIS
LIN {X 62.903,Y -41.245,Z -77.576,A -90.000,B 90.000,C 0.000} C_DIS
LIN {X 63.002,Y -41.250,Z -77.567,A -90.000,B 90.000,C 0.000} C_DIS
LIN {X 63.106,Y -41.255,Z -77.547,A -90.000,B 90.000,C 0.000} C_DIS
LIN {X 63.214,Y -41.261,Z -77.514,A -90.000,B 90.000,C 0.000} C_DIS
LIN {X 63.270,Y -41.264,Z -77.493,A -90.000,B 90.000,C 0.000} C_DIS
LIN {X 63.383,Y -41.270,Z -77.441,A -90.000,B 90.000,C 0.000} C_DIS
LIN {X 63.500,Y -41.277,Z -77.376,A -90.000,B 90.000,C 0.000} C_DIS
LIN {X 63.620,Y -41.283,Z -77.297,A -90.000,B 90.000,C 0.000} C_DIS
LIN {X 63.681,Y -41.287,Z -77.253,A -90.000,B 90.000,C 0.000} C_DIS
LIN {X 63.742,Y -41.290,Z -77.205,A -90.000,B 90.000,C 0.000} C_DIS
LIN {X 63.866,Y -41.298,Z -77.096,A -90.000,B 90.000,C 0.000} C_DIS
LIN {X 64.057,Y -41.308,Z -76.909,A -90.000,B 90.000,C 0.000} C_DIS
LIN {X 64.088,Y -41.310,Z -76.875,A -90.000,B 90.000,C 0.000} C_DIS
LIN {X 64.177,Y -41.315,Z -76.771,A -90.000,B 90.000,C 0.000} C_DIS
LIN {X 64.244,Y -41.320,Z -76.682,A -90.000,B 90.000,C 0.000} C_DIS
LIN {X 64.307,Y -41.324,Z -76.586,A -90.000,B 90.000,C 0.000} C_DIS
LIN {X 64.379,Y -41.329,Z -76.472,A -90.000,B 90.000,C 0.000} C_DIS
LIN {X 64.588,Y -41.342,Z -76.126,A -90.000,B 90.000,C 0.000} C_DIS
LIN {X 64.687,Y -41.341,Z -75.953,A -90.000,B 90.000,C 0.000} C_DIS
LIN {X 64.879,Y -41.308,Z -75.600,A -90.000,B 90.000,C 0.000} C_DIS
LIN {X 65.008,Y -41.283,Z -75.352,A -90.000,B 90.000,C 0.000} C_DIS
LIN {X 65.058,Y -41.271,Z -75.248,A -90.000,B 90.000,C 0.000} C_DIS
LIN {X 65.130,Y -41.246,Z -75.079,A -90.000,B 90.000,C 0.000} C_DIS
LIN {X 65.162,Y -41.229,Z -74.983,A -90.000,B 90.000,C 0.000} C_DIS
LIN {X 65.175,Y -41.212,Z -74.914,A -90.000,B 90.000,C 0.000} C_DIS
LIN {X 65.176,Y -41.206,Z -74.897,A -90.000,B 90.000,C 0.000} C_DIS
LIN {X 65.172,Y -41.195,Z -74.870,A -90.000,B 90.000,C 0.000} C_DIS
LIN {X 65.167,Y -41.190,Z -74.860,A -90.000,B 90.000,C 0.000} C_DIS
LIN {X 65.153,Y -41.179,Z -74.848,A -90.000,B 90.000,C 0.000} C_DIS
LIN {X 65.132,Y -41.169,Z -74.847,A -90.000,B 90.000,C 0.000} C_DIS
LIN {X 65.119,Y -41.164,Z -74.849,A -90.000,B 90.000,C 0.000} C_DIS
LIN {X 65.105,Y -41.163,Z -74.854,A -90.000,B 90.000,C 0.000} C_DIS
LIN {X 65.054,Y -41.176,Z -74.883,A -90.000,B 90.000,C 0.000} C_DIS
LIN {X 64.992,Y -41.195,Z -74.930,A -90.000,B 90.000,C 0.000} C_DIS
LIN {X 64.893,Y -41.225,Z -75.021,A -90.000,B 90.000,C 0.000} C_DIS
LIN {X 64.837,Y -41.241,Z -75.078,A -90.000,B 90.000,C 0.000} C_DIS
LIN {X 64.716,Y -41.273,Z -75.211,A -90.000,B 90.000,C 0.000} C_DIS
LIN {X 64.651,Y -41.287,Z -75.287,A -90.000,B 90.000,C 0.000} C_DIS
LIN {X 64.515,Y -41.313,Z -75.455,A -90.000,B 90.000,C 0.000} C_DIS
LIN {X 64.372,Y -41.329,Z -75.642,A -90.000,B 90.000,C 0.000} C_DIS
LIN {X 64.225,Y -41.334,Z -75.847,A -90.000,B 90.000,C 0.000} C_DIS
LIN {X 64.077,Y -41.327,Z -76.064,A -90.000,B 90.000,C 0.000} C_DIS
LIN {X 63.931,Y -41.317,Z -76.293,A -90.000,B 90.000,C 0.000} C_DIS
LIN {X 63.860,Y -41.312,Z -76.410,A -90.000,B 90.000,C 0.000} C_DIS
LIN {X 63.722,Y -41.302,Z -76.648,A -90.000,B 90.000,C 0.000} C_DIS
LIN {X 63.595,Y -41.289,Z -76.889,A -90.000,B 90.000,C 0.000} C_DIS
LIN {X 63.479,Y -41.271,Z -77.131,A -90.000,B 90.000,C 0.000} C_DIS
LIN {X 63.379,Y -41.255,Z -77.369,A -90.000,B 90.000,C 0.000} C_DIS
LIN {X 63.315,Y -41.244,Z -77.543,A -90.000,B 90.000,C 0.000} C_DIS
LIN {X 63.279,Y -41.237,Z -77.657,A -90.000,B 90.000,C 0.000} C_DIS
LIN {X 63.249,Y -41.231,Z -77.768,A -90.000,B 90.000,C 0.000} C_DIS
LIN {X 63.214,Y -41.222,Z -77.930,A -90.000,B 90.000,C 0.000} C_DIS
LIN {X 63.198,Y -41.215,Z -78.033,A -90.000,B 90.000,C 0.000} C_DIS
LIN {X 63.190,Y -41.207,Z -78.133,A -90.000,B 90.000,C 0.000} C_DIS
LIN {X 63.188,Y -41.199,Z -78.229,A -90.000,B 90.000,C 0.000} C_DIS
LIN {X 63.194,Y -41.191,Z -78.319,A -90.000,B 90.000,C 0.000} C_DIS
LIN {X 63.207,Y -41.184,Z -78.405,A -90.000,B 90.000,C 0.000} C_DIS
LIN {X 63.229,Y -41.178,Z -78.486,A -90.000,B 90.000,C 0.000} C_DIS
LIN {X 63.260,Y -41.174,Z -78.561,A -90.000,B 90.000,C 0.000} C_DIS
LIN {X 63.278,Y -41.172,Z -78.596,A -90.000,B 90.000,C 0.000} C_DIS
LIN {X 63.322,Y -41.171,Z -78.661,A -90.000,B 90.000,C 0.000} C_DIS
LIN {X 63.348,Y -41.171,Z -78.692,A -90.000,B 90.000,C 0.000} C_DIS
LIN {X 63.406,Y -41.173,Z -78.747,A -90.000,B 90.000,C 0.000} C_DIS
LIN {X 63.439,Y -41.176,Z -78.772,A -90.000,B 90.000,C 0.000} C_DIS
LIN {X 63.512,Y -41.191,Z -78.817,A -90.000,B 90.000,C 0.000} C_DIS
LIN {X 63.596,Y -41.207,Z -78.853,A -90.000,B 90.000,C 0.000} C_DIS
LIN {X 63.691,Y -41.223,Z -78.882,A -90.000,B 90.000,C 0.000} C_DIS
LIN {X 63.742,Y -41.232,Z -78.893,A -90.000,B 90.000,C 0.000} C_DIS
LIN {X 63.854,Y -41.250,Z -78.908,A -90.000,B 90.000,C 0.000} C_DIS
LIN {X 63.978,Y -41.268,Z -78.915,A -90.000,B 90.000,C 0.000} C_DIS
LIN {X 64.114,Y -41.288,Z -78.911,A -90.000,B 90.000,C 0.000} C_DIS
LIN {X 64.262,Y -41.308,Z -78.898,A -90.000,B 90.000,C 0.000} C_DIS
LIN {X 64.316,Y -41.316,Z -78.892,A -90.000,B 90.000,C 0.000} C_DIS
LIN {X 64.439,Y -41.332,Z -78.872,A -90.000,B 90.000,C 0.000} C_DIS
LIN {X 64.604,Y -41.354,Z -78.832,A -90.000,B 90.000,C 0.000} C_DIS
LIN {X 64.802,Y -41.380,Z -78.764,A -90.000,B 90.000,C 0.000} C_DIS
LIN {X 64.917,Y -41.394,Z -78.713,A -90.000,B 90.000,C 0.000} C_DIS
LIN {X 64.974,Y -41.401,Z -78.684,A -90.000,B 90.000,C 0.000} C_DIS
LIN {X 65.051,Y -41.410,Z -78.641,A -90.000,B 90.000,C 0.000} C_DIS
LIN {X 65.119,Y -41.415,Z -78.600,A -90.000,B 90.000,C 0.000} C_DIS
LIN {X 65.222,Y -41.423,Z -78.531,A -90.000,B 90.000,C 0.000} C_DIS
LIN {X 65.345,Y -41.432,Z -78.434,A -90.000,B 90.000,C 0.000} C_DIS
LIN {X 65.466,Y -41.440,Z -78.322,A -90.000,B 90.000,C 0.000} C_DIS
LIN {X 65.511,Y -41.443,Z -78.276,A -90.000,B 90.000,C 0.000} C_DIS
LIN {X 65.614,Y -41.448,Z -78.161,A -90.000,B 90.000,C 0.000} C_DIS
LIN {X 65.720,Y -41.453,Z -78.036,A -90.000,B 90.000,C 0.000} C_DIS
LIN {X 65.805,Y -41.456,Z -77.926,A -90.000,B 90.000,C 0.000} C_DIS
LIN {X 65.903,Y -41.460,Z -77.790,A -90.000,B 90.000,C 0.000} C_DIS
LIN {X 65.993,Y -41.462,Z -77.653,A -90.000,B 90.000,C 0.000} C_DIS
LIN {X 66.084,Y -41.459,Z -77.509,A -90.000,B 90.000,C 0.000} C_DIS
LIN {X 66.203,Y -41.448,Z -77.314,A -90.000,B 90.000,C 0.000} C_DIS
LIN {X 66.325,Y -41.431,Z -77.113,A -90.000,B 90.000,C 0.000} C_DIS
LIN {X 66.431,Y -41.408,Z -76.930,A -90.000,B 90.000,C 0.000} C_DIS
LIN {X 66.507,Y -41.385,Z -76.790,A -90.000,B 90.000,C 0.000} C_DIS
LIN {X 66.636,Y -41.334,Z -76.554,A -90.000,B 90.000,C 0.000} C_DIS
LIN {X 66.696,Y -41.308,Z -76.435,A -90.000,B 90.000,C 0.000} C_DIS
LIN {X 66.696,Y -60.000,Z -76.435,A -90.000,B 90.000,C 0.000} C_DIS
LIN {X 47.456,Y -60.000,Z -55.201,A -90.000,B 90.000,C 0.000} C_DIS
LIN {X 47.456,Y -41.308,Z -55.201,A -90.000,B 90.000,C 0.000} C_DIS
LIN {X 47.585,Y -41.370,Z -55.289,A -90.000,B 90.000,C 0.000} C_DIS
LIN {X 47.820,Y -41.476,Z -55.442,A -90.000,B 90.000,C 0.000} C_DIS
LIN {X 48.000,Y -41.480,Z -55.427,A -90.000,B 90.000,C 0.000} C_DIS
LIN {X 48.184,Y -41.482,Z -55.418,A -90.000,B 90.000,C 0.000} C_DIS
LIN {X 48.320,Y -41.485,Z -55.416,A -90.000,B 90.000,C 0.000} C_DIS
LIN {X 49.310,Y -41.480,Z -55.417,A -90.000,B 90.000,C 0.000} C_DIS
LIN {X 49.862,Y -41.479,Z -55.420,A -90.000,B 90.000,C 0.000} C_DIS
